// TwinCAT 3 PLC project smarAct
// Title: ESO LDC SmarAct Library
// Company: ESO
// Author: Dan Popovic
// ProjectVersion: 0.0.2.1
// Description: Local Device Control - LDC SmarAct Library based on State Machine.
// ProgramVersion: 3.1.4023.0
// libraries:
//   ESO LDC Comm Common Library, * (ESO)
//   ESO LDC Comm Tcp Library, * (ESO)
//   Tc2_Standard, * (Beckhoff Automation GmbH)
//   Tc2_System, * (Beckhoff Automation GmbH)
//   Tc2_TcpIp, * (Beckhoff Automation GmbH)
//   Tc2_Utilities, * (Beckhoff Automation GmbH)
//   Tc3_Module, * (Beckhoff Automation GmbH)
//   VisuDialogs, * (System)
//   VisuSymbols,3.5.10.0,System
// project tree:
//   DUTs/Enumerated/ E_SA_CH_ERROR.TcDUT, E_SA_RPC_ERROR.TcDUT, E_SA_POS_ELT_STATE.TcDUT, E_SA_POS_ELT_SUBSTATE.TcDUT, E_SA_CH_CMD.TcDUT, E_SA_CH_STATE.TcDUT, E_SA_CMD_TYPE.TcDUT, E_SA_DEV_STATE.TcDUT, E_SA_MOD_STATE.TcDUT, E_SA_POS_SM_STATE.TcDUT
//   DUTs/Simulation/ E_SA_SIM_CH_SM_STATE.TcDUT, T_SA_SIM_CH_CFG.TcDUT, T_SA_SIM_CH_CTRL.TcDUT, T_SA_SIM_CH_STATUS.TcDUT
//   DUTs/Structures/ T_SA_CFG.TcDUT, T_SA_CH_CFG.TcDUT, T_SA_CH_CTRL.TcDUT, T_SA_CH_STATUS.TcDUT, T_SA_CH_STATE.TcDUT, T_SA_COMMAND.TcDUT, T_SA_CTRL.TcDUT, T_SA_DEV_STATUS.TcDUT, T_SA_MOD_STATE.TcDUT, T_SA_DEV_STATE.TcDUT, T_SA_STATUS.TcDUT
//   Examples/ FB_SA_CH_PDS_IRIS.TcPOU, FB_SMARACT_SIM.TcPOU, FB_SMARACT_PDS.TcPOU
//   / GlobalTextList.TcGTLO, PlcTask.TcTTO, Visualization Manager.TcVMO (not stored)
//   POUs/ FB_SMAR_ACT_BASE.TcPOU, FB_SA_CHANNEL_BASE.TcPOU, F_GetRpcErrorText.TcPOU, F_STRING_TO_LINT.TcPOU, MAIN.TcPOU
//   POUs/Simulation/ FB_SIM_SA_CHANNEL.TcPOU, FB_SIM_SMAR_ACT.TcPOU
//   Version/ Global_Version.TcGVL
//   VISUs/GUIs/ GUI_SmarAct_PDS.TcVIS, GUI_SmarAct_SIM.TcVIS
//   VISUs/Templates/ GUI_TEMPLATE_SMAR_ACT.TcVIS
// real-time tasks:
//   TASK PlcTask: cycle T#1ms, priority 20, ADS port 350
// I/O:
//   DEVICE Device 1 (EtherCAT), AmsNetId 134.171.12.217.2.1
//     Term 1 (EK1200) [EK1200-5000 EtherCAT Power supply (2A E-Bus)]
//       Term 2 (EL6002) [EL6002 Interface 2Ch. (RS232)]
//       Term 3 (EK1110) [EK1110 EtherCAT extension]
//     Term 4 (EK1100) [EK1100 EtherCAT Coupler (2A E-Bus)]
//       Term 5 (EL3068) [EL3068 8Ch. Ana. Input 0-10V]
//       Term 6 (EL4008) [EL4008 8Ch. Ana. Output 0-10V, 12bit]
//       Term 7 (EL2008) [EL2008 8Ch. Dig. Output 24V, 0.5A]
//       Term 8 (EL1008) [EL1008 8Ch. Dig. Input 24V, 3ms]
//       Term 9 (EL3202) [EL3202 2Ch. Ana. Input PT100 (RTD)]
//       Term 10 (EL6614) [EL6614 4 Port Switch (Ethernet, CoE)]
//       Term 11 (EL6688) [EL6688 - External Synchronisation Interface (IEEE1588)]
//       Term 12 (EL9011) [EL9011 End Terminal]
// variable links:
//   smarAct/smarAct Instance <-> Device 1 (EtherCAT)/Term 4 (EK1100)/Term 10 (EL6614)
//     PlcTask Inputs/MAIN.SIM_SA.Device.i_nCouplerState <-> InfoData/State
//     PlcTask Inputs/MAIN.SmarAct_PDS.comm.i_nCouplerState <-> InfoData/State
//     PlcTask Inputs/MAIN.SmarAct_Sim.comm.i_nCouplerState <-> InfoData/State
//   smarAct/smarAct Instance <-> Device 1 (EtherCAT)/Term 4 (EK1100)/Term 8 (EL1008)
//     PlcTask Inputs/MAIN.i_bDummy <-> Channel 1/Input

CONFIGURATION smarAct
    RESOURCE PLC ON TwinCAT3
        TASK PlcTask(INTERVAL := T#1ms, PRIORITY := 20);
        PROGRAM MAIN WITH PlcTask : MAIN;
    END_RESOURCE
END_CONFIGURATION

// ---- DUTs/Enumerated/E_SA_CH_ERROR.TcDUT
{attribute 'qualified_only'}
// 'strict' cannot be used since we mix our own codes with TC codes
//{attribute 'strict'}
TYPE E_SA_CH_ERROR :
(
	OK				:= 0,
	HW_NOT_OP,
	CONFIG,				// Configuration problem, e.g. pointers not set.		
	LOCAL,			
	SETPOS,
	STOP,
	
	ABORT,
	SW_LIMIT_LOWER,
	SW_LIMIT_UPPER,
	ENABLE,
	CTRL,				// MCS2 controller error
	COMM				// MCS2 controller communication problem

);
END_TYPE

// ---- DUTs/Enumerated/E_SA_RPC_ERROR.TcDUT
{attribute 'qualified_only'}
//{attribute 'strict'}
TYPE E_SA_RPC_ERROR :
(
	OK						:= 0,
	NOT_OP					:= -1,			
	NOT_NOTOP_READY			:= -2,			
	NOT_NOTOP_NOTREADY		:= -3,			
	LOCAL					:= -4,			
	SW_LIMIT_LOWER			:= -5,			
	SW_LIMIT_UPPER			:= -6,			
	CHANNEL					:= -7,			
	VEL_ZERO				:= -8,			
	VEL_NEG					:= -9,			
	VEL_MAX					:= -10,			
	CH_NOT_OP				:= -11,
	CTRL_ERROR				:= -12,
	MOVING					:= -13,
	COMM					:= -14	// MCS2 Controller communication problem			
);
END_TYPE

// ---- DUTs/Enumerated/E_SA_POS_ELT_STATE.TcDUT
{attribute 'qualified_only'}
{attribute 'strict'}
TYPE E_SA_POS_ELT_STATE :
(
	NONE	:= 0,
	NOTOP,
	OP
);
END_TYPE

// ---- DUTs/Enumerated/E_SA_POS_ELT_SUBSTATE.TcDUT
{attribute 'qualified_only'}
{attribute 'strict'}
TYPE E_SA_POS_ELT_SUBSTATE :
(
	NONE					:= 0,
	
	NOTOP_NOTREADY			:= 100,
	NOTOP_READY				:= 101,
	NOTOP_INITIALIZING		:= 102,
	NOTOP_ABORTING			:= 107,
	
	NOTOP_ERROR				:= 199,
	
	
	OP_STANDSTILL			:= 216,            
	OP_MOVING				:= 217,
	OP_SETTING_POS			:= 218,
	OP_STOPPING				:= 219,
	
	OP_ERROR				:= 299
);
END_TYPE

// ---- DUTs/Enumerated/E_SA_CH_CMD.TcDUT
{attribute 'qualified_only'}
{attribute 'strict'}
TYPE E_SA_CH_CMD :
(
	NONE	:= 0,
	RESET,
	CALIB,
	REF,
	ENABLE,
	DISABLE,
	STOP,
	MOV
);
END_TYPE

// ---- DUTs/Enumerated/E_SA_CH_STATE.TcDUT
{attribute 'qualified_only'}
{attribute 'strict'}
TYPE E_SA_CH_STATE :
(
	BIT_ACTIVELY_MOVING			:=	16#00000001,
	BIT_CLOSED_LOOP_ACTIVE		:=	16#00000002,
	BIT_CALIBRATING				:=	16#00000004,
	BIT_REFERENCING				:=	16#00000008,
	BIT_MOVE_DELAYED			:=	16#00000010,
	BIT_SENSOR_PRESENT			:=	16#00000020,
	BIT_IS_CALIBRATED			:=	16#00000040,
	BIT_IS_REFERENCED			:=	16#00000080,
	BIT_END_STOP_REACHED		:=	16#00000100,
	BIT_RANGE_LIMIT_REACHED		:=	16#00000200,
	BIT_FOLLOWING_LIMIT_REACHED	:=	16#00000400,
	BIT_MOVEMENT_FAILED			:=	16#00000800,
	BIT_IS_STREAMING			:=	16#00001000,
	BIT_POSITIONER_OVERLOAD		:=	16#00002000,
	BIT_OVER_TEMPERATURE		:=	16#00004000,
	BIT_REFERENCE_MARK			:=	16#00008000,
	BIT_IS_PHASED				:=	16#00010000,
	BIT_POSITIONER_FAULT		:=	16#00020000,
	BIT_AMPLIFIER_ENABLED		:=	16#00040000,
	BIT_IN_POSITION				:=	16#00080000
) UDINT;
END_TYPE

// ---- DUTs/Enumerated/E_SA_CMD_TYPE.TcDUT
{attribute 'qualified_only'}
{attribute 'strict'}
TYPE E_SA_CMD_TYPE :
(
	INIT := 0,	// Commands for system initialisation
	READ,		// Commands for Reading status
	CFG,		// Commands for Configuring channels
	CTRL		// Commands for Controlling positioners, e.g. CAL, REF, MOVE, STOP
);
END_TYPE

// ---- DUTs/Enumerated/E_SA_DEV_STATE.TcDUT
{attribute 'qualified_only'}
{attribute 'strict'}
TYPE E_SA_DEV_STATE :
(
	BIT_HM_PRESENT				:= 16#00000001,
	BIT_MOVEMENT_LOCKED			:= 16#00000002,
	BIT_AMPLIFIER_LOCKED		:= 16#00000004,
	BIT_IO_MODULE_INPUT			:= 16#00000008,
	BIT_GLOBAL_INPUT			:= 16#00000010,
	BIT_INTERNAL_COMM_FAILURE	:= 16#00000100,
	BIT_IS_STREAMING			:= 16#00001000
) UDINT;
END_TYPE

// ---- DUTs/Enumerated/E_SA_MOD_STATE.TcDUT
{attribute 'qualified_only'}
{attribute 'strict'}
TYPE E_SA_MOD_STATE :
(
	BIT_SM_PRESENT				:= 16#00000001,
	BIT_BOOSTER_PRESENT			:= 16#00000002,
	BIT_ADJUSTMENT_ACTIVE		:= 16#00000004,
	BIT_IOM_PRESENT				:= 16#00000008,
	BIT_INTERNAL_COMM_FAILURE	:= 16#00000100,
	BIT_FAN_FAILURE				:= 16#00000800,
	BIT_POWER_SUPPLY_FAILURE	:= 16#00001000,
	BIT_POWER_SUPPLY_OVERLOAD	:= 16#00002000,
	BIT_OVER_TEMPERATURE		:= 16#00004000
) UDINT;
END_TYPE

// ---- DUTs/Enumerated/E_SA_POS_SM_STATE.TcDUT
{attribute 'qualified_only'}
{attribute 'strict'}
TYPE E_SA_POS_SM_STATE :
(
	// Positioner State Machine States
	NOT_READY := 0,	// The system just started.
	CALIB,			// The Positioner is Calibrating
	INIT,			// The Positioner is INITialising/REFerencing
	POST_INIT,		// In POST_INIT we calibrate REF and read CFG once.
	CALIB_REF,		// Calibrate REF position.
	READY,			// NOT OPERATIONAL / READY (i.e. REFerenced)
	
	OP,				// Positioner is Operational
	MOVING,			// Positioner is moving
	STOP,			// Positioner is stopping
	ERROR			// Positioner is in error
);
END_TYPE

// ---- DUTs/Simulation/E_SA_SIM_CH_SM_STATE.TcDUT
{attribute 'qualified_only'}
{attribute 'strict'}
TYPE E_SA_SIM_CH_SM_STATE :
(
	IDLE := 0,
	CALIB,
	REF,
	MOV,
	STOP
);
END_TYPE

// ---- DUTs/Simulation/T_SA_SIM_CH_CFG.TcDUT
TYPE T_SA_SIM_CH_CFG :
STRUCT
	
	//
	// SmarAct Positioner configuration parameters.
	// All units are Positioner System Units [DevU], pd and nm.
	//
	
	//
	// Channel Number [0..17]
	//
	nCHAN:			UINT := 0;

	//
	// MODule number that the channel belongs to [0..5].
	//
	nMOD:			UINT;	// Module  number [0..5]

	nCLIN:			DINT := 1;	// Channel Control Loop Input (1 = SENSOR)

	nBASE_UNIT:		DINT := 2;	// Channel Base Unit (2=meter, 3=degree)

	nBASE_RES:		DINT := -9;	// Channel Base Resolution

	nTUN_MTYP:		DINT := 0;	// Channel Positioner Movement Type (0=linear, 1=rotary)

	nTUN_RTYP:		DINT := 2;	// Channel Positioner Reference Type (1=end stop, 2=single coded)

	//
	// Positioning
	//

	// Position of Reference [UU].
	// This is the position to set for the REFerence (INIT).
	// Equivalent to 'Calibrate on Switch' in FB_MOTOR.
	// ':CHAN#:POS <pos>'	
	//
	lnREF_POS:		LINT := 0;
	
	lnREF_VEL:		LINT := 1;	// Velocity for referencing DevU/s]

	lnVEL:			LINT := 1;	// Velocity for referencing DevU/s]
	
	// Hold Time [ms].
	// In-position holding time. (-1) means indefinite.
	// ':CHAN#:HOLD <time>'
	//
	nHOLD:			DINT := -1;
	

	
	// In Position Threshold in [UU].
	// ':CHAN#:INP:THR <thr>'
	//
	nINP_THR:		UDINT := 1;	
	
	// In Position Delay [ms]
	// ':CHAN#:INP:DEL <delay>'
	// Move is complete after the positioner has been in position for <delay> ms.
	//
	nINP_DEL:		UDINT := 1000;
	
	// Range Limit Min (lower limit) [UU].
	// ':CHAN#:RLIM:MIN <lim>'
	// Note: If both lrRangeLimitMin and lrRangeLimitMax are set to 0.0,
	//       limits are not set.
	//
	lnRLIM_MIN:		LINT := 0;

	// Range Limit Max (upper limit) [UU].
	// ':CHAN#:RLIM:MAX <lim>'
	//
	lnRLIM_MAX:		LINT := 0;


	//
	// Calibration, Referencing (INIT) and State configuration
	//
	
	// Referencing Options.
	// :CHAN#:REF:OPT <opt>
	// It is expected that only the direction for referencing is needed to be configured.
	//    0 – positive (default)
	//    1 - negative
	nREF_OPT:		UINT := 0;

	// Calibration Options.
	// :CHAN#:CAL:OPT <opt>
	// It is expected that only the direction for Calibration is needed to be configured.
	//    0 – positive (default)
	//    1 - negative
	nCAL_OPT:		UINT := 0;

	// Positionign control options.
	// 256 - ‘In Position’ flag is set on move completion.
	// ':CHAN#:PCON:OPT <opt>'
	nPCON_OPT:		UINT := 256;
	
	
	
END_STRUCT
END_TYPE

// ---- DUTs/Simulation/T_SA_SIM_CH_CTRL.TcDUT
TYPE T_SA_SIM_CH_CTRL :
STRUCT
	
	nMode:	DINT := 0;		// Movement type: 0 - Absolute, 1 - Relative. 
	lnPOS:	LINT;			// Position in Positioner/Device Units, i.e. [nd] or [pm]
	lnVEL:	LINT := 1000;	// Velocity in Positioner/Device, i.e. [nd/s] or [pm/s]
	
END_STRUCT
END_TYPE

// ---- DUTs/Simulation/T_SA_SIM_CH_STATUS.TcDUT
TYPE T_SA_SIM_CH_STATUS :
STRUCT
	//
	// Positioner State Machine State.
	// Depending on the State, different command sets will be executed.
	//
	nPosState:			E_SA_POS_SM_STATE := E_SA_POS_SM_STATE.NOT_READY;
	

	//
	// Channel Configuration parameters read from the controller.
	// A channel is a Positioner.
	//
	nCLIN:				DINT;			// Control Loop Input, 1-SENSOR
	nTUN_BASE_UNIT:		DINT;			// Positioner Base Unit, 2-meter, 3-degree
	nTUN_BASE_RES:		DINT;			// Positioner Base Resolution, 1x10-9 or 1x10-12
	nTUN_MTYP:			DINT;			// Positioner Movement Type, 0-linear, 1-rotation, etc
	nTUN_RTYP:			DINT;			// Positioner Reference Type, 2-SINGLE_CODED


	lnPosTarget:		LINT;			// Target  position in Positioner Units
	lnPosActual:		LINT;			// Current position in Positioner Units
	lnPosStart:			LINT;			// Starting position for MOVE in Positioner Units
	lnDistance:			LINT := 0;		// move distance


	bConfigured:		BOOL;			// Flag if M_Configure has been executed.	
	bError:				BOOL;
	bInitialised:		BOOL;			// Flag if positioner has been initialised/referenced

	//
	// Channel State parameters read from the controller
	// A channel is a Positioner.
	//
	nSTATE:				UDINT;			// Positioner State as UDINT
	stState:			T_SA_CH_STATE;	// Positioner State structure, from nSTATE
	
END_STRUCT
END_TYPE

// ---- DUTs/Structures/T_SA_CFG.TcDUT
TYPE T_SA_CFG EXTENDS T_RS_BASE_CFG:
STRUCT
	//
	// INIT commands.
	// Executed during Initialisation, before going to OPERATIONAL.
	//
	{attribute 'OPC.UA.DA' := '0'}
	cmdList_Init:	ARRAY [0..7] OF T_SA_COMMAND := [
							(cmd := '*IDN?', 			nReplies := 1),
							(cmd := ':DEV:SNUM?', 		nReplies := 1),
							(cmd := ':DEV:STAT?', 		nReplies := 1),
							(cmd := '', 		nReplies := 0),
							(cmd := '', 		nReplies := 0),
							(cmd := '', 		nReplies := 0),
							(cmd := '', 		nReplies := 0),
							(cmd := '', 		nReplies := 0)];

	//
	// List of commands to SET Channel/Positioner Configuration.
	// Note the # and *** characters !!!
	// The actual command will be set like this:
	//    #   will be replaced with channel number
	//    *** will be replaced with a value
	// Example:
	//    ':CHAN#:PCON:OPT ***' => ':CHAN1:PCON:OPT 256'
	//
	// Important NOTE:
	// At this stage RLIM:MIN and RLIM:MAX are disabled, i.e. = 0.
	// The actual limits will be set at the E_SA_POS_SM_STATE.CALIB_REF stage,
	// see M_SetCmdList().
	//
	// These commands are sent only once, just before the positioner is 
	// commanded to Reference (INIT).
	//
	{attribute 'OPC.UA.DA' := '0'}
	cmdList_CfgSet:	ARRAY [0..15] OF T_SA_COMMAND := [
							(cmd := ':CHAN#:CAL:OPT ***', 		nReplies := 0),
							(cmd := ':CHAN#:REF:OPT ***', 		nReplies := 0),
							(cmd := ':CHAN#:PCON:OPT ***', 		nReplies := 0),
							(cmd := ':CHAN#:HOLD ***', 			nReplies := 0),
							(cmd := ':CHAN#:INP:THR ***', 		nReplies := 0),
							(cmd := ':CHAN#:INP:DEL ***', 		nReplies := 0),
							(cmd := ':CHAN#:RLIM:MIN 0', 		nReplies := 0),
							(cmd := ':CHAN#:RLIM:MAX 0', 		nReplies := 0),
							(cmd := ':CHAN#:VEL ***', 			nReplies := 0),
							(cmd := ':REF#', 					nReplies := 0),
							(cmd := '', 		nReplies := 0),
							(cmd := '', 		nReplies := 0)];
							

	//				
	// List of commands to GET Channel/Positioner Configuration.
	// These commands are sent from the moment the SW started till the positioner 
	// has been Calibrated or Referenced (INIT).
	// Once the Positioer is Ready, these commans are not sent any more.
	//
	{attribute 'OPC.UA.DA' := '0'}
	cmdList_POST_INIT:	ARRAY [0..15] OF T_SA_COMMAND := [
							(cmd := ':MOD#:STAT?', 			nReplies := 1),
							(cmd := ':CHAN#:STAT?', 		nReplies := 1),
							(cmd := ':CHAN#:CAL:OPT?', 		nReplies := 1),
							(cmd := ':CHAN#:REF:OPT?', 		nReplies := 1),
							(cmd := ':CHAN#:PCON:OPT?', 	nReplies := 1),
							(cmd := ':CHAN#:INP:THR?', 		nReplies := 1),
							(cmd := ':CHAN#:INP:DEL?', 		nReplies := 1),
							(cmd := ':CHAN#:RLIM:MIN?', 	nReplies := 1),
							(cmd := ':CHAN#:RLIM:MAX?', 	nReplies := 1),
							(cmd := ':CHAN#:POS:TARG?', 	nReplies := 1),
							(cmd := ':CHAN#:POS:CURR?', 	nReplies := 1),
							(cmd := '', 		nReplies := 0),
							(cmd := '', 		nReplies := 0),
							(cmd := '', 		nReplies := 0),
							(cmd := '', 		nReplies := 0),
							(cmd := '', 		nReplies := 0)];
							

	//
	// List of Monitoring commands in PRE-OPERATION.
	// Executed before the Positioner has been Referenced/initialised.
	//
	{attribute 'OPC.UA.DA' := '0'}
	cmdList_NOT_READY:	ARRAY [0..15] OF T_SA_COMMAND := [
							(cmd := ':MOD#:STAT?', 			nReplies := 1),
							(cmd := ':CHAN#:STAT?', 		nReplies := 1),
							(cmd := ':CHAN#:POS:TARG?', 	nReplies := 1),
							(cmd := ':CHAN#:POS:CURR?', 	nReplies := 1),
							(cmd := ':CHAN#:PCON:OPT?', 	nReplies := 1),
							(cmd := ':CHAN#:CLIN?', 		nReplies := 1),
							(cmd := ':CHAN#:TUN:BASE:UNIT?',nReplies := 1),
							(cmd := ':CHAN#:TUN:BASE:RES?', nReplies := 1),
							(cmd := ':CHAN#:TUN:MTYP?', 	nReplies := 1),
							(cmd := ':CHAN#:TUN:RTYP?', 	nReplies := 1),
							(cmd := ':CHAN#:INP:THR?', 		nReplies := 1),
							(cmd := ':CHAN#:INP:DEL?', 		nReplies := 1),
							(cmd := ':CHAN#:RLIM:MIN?', 	nReplies := 1),
							(cmd := ':CHAN#:RLIM:MAX?', 	nReplies := 1),
							(cmd := '', 		nReplies := 0),
							(cmd := '', 		nReplies := 0)];
			

	//
	// List of Monitoring commands in OPERATION.
	// Executed once the Positioner has been Referenced/initialised.
	//
	{attribute 'OPC.UA.DA' := '0'}
	cmdList_Mon:	ARRAY [0..15] OF T_SA_COMMAND := [
							(cmd := ':MOD#:STAT?', 			nReplies := 1),
							(cmd := ':CHAN#:STAT?', 		nReplies := 1),
							(cmd := ':CHAN#:POS:TARG?', 	nReplies := 1),
							(cmd := ':CHAN#:POS:CURR?', 	nReplies := 1),
							(cmd := '', 		nReplies := 0),
							(cmd := '', 		nReplies := 0),
							(cmd := '', 		nReplies := 0),
							(cmd := '', 		nReplies := 0),
							(cmd := '', 		nReplies := 0),
							(cmd := '', 		nReplies := 0),
							(cmd := '', 		nReplies := 0),
							(cmd := '', 		nReplies := 0),
							(cmd := '', 		nReplies := 0),
							(cmd := '', 		nReplies := 0),
							(cmd := '', 		nReplies := 0),
							(cmd := '', 		nReplies := 0)];
			

	//
	// Array of used channels. Set to TRUE for each used channel.
	// 18 channels max. 6 modules [0..5], 3 connections each [CH1, CH2, CH3].
	// channel = (Module x 3) + (CH-1)
	// For example:
	//   First connection (CH1) of first module (Module0): channel = 0 x 3 + (1-1) = 0
	//   Second connection (CH2) of first module (Module0): channel = 0 x 3 + (2-1) = 1
	//   Third connection (CH3) of third module (Module2): channel = 2 x 3 + (3-1) = 8
	//  
	arrUsedCh:	ARRAY [0..17] 	OF BOOL;	

	//
	// Array of used modules. Set to TRUE for each used module.
	// Automatically populated in method M_Configure().
	//
	arrUsedMod:	ARRAY [0..5] 	OF BOOL;	
	
	// Channel configuration structures
//	arrChCfg:	ARRAY [0..17] OF T_SA_CH_CFG;

END_STRUCT
END_TYPE

// ---- DUTs/Structures/T_SA_CH_CFG.TcDUT
TYPE T_SA_CH_CFG :
STRUCT
	sName:	STRING := 'Not Used';	// Positioner name, e.g. 'PYR Filter Wheel'
	sUnits:	STRING := 'none';		// Positioner User Units
	
	bUsed:	BOOL;
	
	lrMaxVelocity:	LREAL := 1.0;	// Maximum velocity	[UU]
	
	//
	// SmarAct Positioner configuration parameters.
	// All units are User Units [UU], mm, deg, etc.
	// The driver converts them into Positioner units.
	// During Referencing (INIT), these parameters will be written to
	// the positioner.
	// The monitoring task will read them from the positioner and 
	// save them into T_SA_CH_STATUS that is contained in T_SA_STATUS.
	//
	
	//
	// Channel Number [0..17]
	//
	// 18 channels max. 6 modules [0..5], 3 connections each [CH1, CH2, CH3].
	// channel = (Module x 3) + (CH-1)
	// For example:
	//   First connection (CH1) of first module (Module0): channel = 0 x 3 + (1-1) = 0
	//   Second connection (CH2) of first module (Module0): channel = 0 x 3 + (2-1) = 1
	//   Third connection (CH3) of third module (Module2): channel = 2 x 3 + (3-1) = 8
	//  
	nCHAN:			UINT := 0;

	//
	// MODule number that the channel belongs to [0..5].
	// Calculated from the channel number. i.e. the index of this instance.
	// channel = (Module x 3) + (CH-1)
	// Module = index / 3
	// index = 0, 1 or 2    => Module = 0
	// index = 3, 4 or 5    => Module = 1
	// ...
	// index = 15, 16 or 17 => Module = 5
	//
	nMOD:			UINT;	// Module  number [0..5]

	//
	// Positioning
	//

	// Conversion from UU to SmarAct units, i.e. [nd] or [pm].
	// This is just the correction of the Base Resolution (if needed).
	// Pos [SmarAct] = lnScale * Pos [UU] / EXPT(10, T_SA_CH_STATUS:nTUN_BASE_RES)
	//
	lrScale:		LREAL := 1.0;	
	
	
	// Position of Reference [UU].
	// This is the position to set for the REFerence (INIT).
	// Equivalent to 'Calibrate on Switch' in FB_MOTOR.
	// Set position for Reference in User Units
	// ':CHAN#:POS <pos>'	
	// <pos> = lrREF_POS  / EXPT(10, T_SA_CH_STATUS:nTUN_BASE_RES) * lnScale
	//
	lrREF_POS:		LREAL := 0;
	
	lrREF_VEL:		LREAL := 0.01;	// Velocity for referencing [UU/s]
	
	// Hold Time [ms].
	// In-position holding time. (-1) means indefinite.
	// ':CHAN#:HOLD <time>'
	//
	nHOLD:			DINT := -1;
	
	
	
	// In Position Threshold in [UU].
	// ':CHAN#:INP:THR <thr>'
	//
	lrINP_THR:		LREAL := 0.01;	
	
	// In Position Delay [ms]
	// ':CHAN#:INP:DEL <delay>'
	// Move is complete after the positioner has been in position for <delay> ms.
	//
	nINP_DEL:		UDINT := 1000;
	
	// Range Limit Min (lower limit) [UU].
	// ':CHAN#:RLIM:MIN <lim>'
	// Note: If both lrRangeLimitMin and lrRangeLimitMax are set to 0.0,
	//       limits are not set.
	//
	lrRangeLimitMin:	LREAL := 0.0;

	// Range Limit Max (upper limit) [UU].
	// ':CHAN#:RLIM:MAX <lim>'
	//
	lrRangeLimitMax:	LREAL := 0.0;
	
	
	//
	// Calibration, Referencing (INIT) and State configuration
	//
	
	// Referencing Options.
	// :CHAN#:REF:OPT <opt>
	// It is expected that only the direction for referencing is needed to be configured.
	//    0 – positive (default)
	//    1 - negative
	nREF_OPT:		UINT := 0;

	// Calibration Options.
	// :CHAN#:CAL:OPT <opt>
	// It is expected that only the direction for Calibration is needed to be configured.
	//    0 – positive (default)
	//    1 - negative
	nCAL_OPT:		UINT := 0;

	// Positionign control options.
	// 256 - ‘In Position’ flag is set on move completion.
	// ':CHAN#:PCON:OPT <opt>'
	nPCON_OPT:		UINT := 256;
	
	
	
END_STRUCT
END_TYPE

// ---- DUTs/Structures/T_SA_CH_CTRL.TcDUT
TYPE T_SA_CH_CTRL :
STRUCT
	//
	// Control structure for a single channel/positioner.
	//
	
	//
	// Active command.
	// Setting nCmd to something other than NONE will
	// trigger execution of commands REF, STOP, MOV.
	//
	nCmd:	E_SA_CH_CMD := E_SA_CH_CMD.NONE;	// Active command

	lrPos:	LREAL;		// Position in User Units, i.e. [deg] or [mm]
	lrOff:	LREAL;		// Position offset in User Units, i.e. [deg] or [mm]
	lrVel:	LREAL;		// Velocity in User Units, i.e. [deg/s] or [mm/sec]
	
END_STRUCT
END_TYPE

// ---- DUTs/Structures/T_SA_CH_STATUS.TcDUT
TYPE T_SA_CH_STATUS :
STRUCT
	bLocal:			BOOL	:= FALSE;	// if TRUE, device operated from PLC GUI 

	nErrorCode: 	E_SA_CH_ERROR 	:= E_SA_CH_ERROR.OK;	// Error code 
	nRpcErrorCode: 	E_SA_RPC_ERROR 	:= E_SA_RPC_ERROR.OK;	// RPC Error code

	bCtrlCommProblem:	BOOL;			// SmarAct MCS2 Controller Comm Problem
	nCtrlErrorCode: E_SM_ERROR;			// SmarAct MCS2 Controller Error code
	nCtrlState:		E_RS_BASE_STATE;	// SmarAct MCS2 Controller State	

	sErrorText: 	STRING 	:= 'OK'; 			// Error text 
	sRpcErrorText: 	STRING 	:= 'OK'; 			// RPC Error text 
	sStatus: 		STRING 	:= 'OK'; 			// Status in textual form, e.g. 'OFF' 
	
	//
	// Standard ELT States and Substates
	//
	nState:			E_SA_POS_ELT_STATE 		:= E_SA_POS_ELT_STATE.NOTOP;
	nSubstate:		E_SA_POS_ELT_SUBSTATE	:= E_SA_POS_ELT_SUBSTATE.NOTOP_NOTREADY;
	
	sState:			STRING	:= 'NOTOP';
	sSubstate:		STRING	:= 'NOT READY';

	//
	// Positioner State Machine State.
	// Depending on the State, different command sets will be executed.
	//
	nPosState:			E_SA_POS_SM_STATE := E_SA_POS_SM_STATE.NOT_READY;
	nLastPosState:		E_SA_POS_SM_STATE := E_SA_POS_SM_STATE.NOT_READY;
	

	lrPosTarget:		LREAL;			// Target  position in User Units
	lrPosActual:		LREAL;			// Current position in User Units

	bConfigured:		BOOL;			// Flag if M_Configure has been executed.	
	bError:				BOOL;
	bEnabled:			BOOL;			// Flag if axis is enabled
	bInitialised:		BOOL;			// Flag if positioner has been initialised/referenced
	bInPosition:		BOOL;			// Flag if axis is In-Position

	//
	// Channel State parameters read from the controller
	// A channel is a Positioner.
	//
	nCH_STATE:				UDINT;			// Positioner State as UDINT
	{attribute 'OPC.UA.DA' := '0'}
	stState:			T_SA_CH_STATE;	// Positioner State structure, from nSTATE
	
	//
	// Device/Channel/Positioner status in user units, i.e. [pm] and [nd].
	// These values are read periodically.
	// Values are normally huge, e.g. pos=18000000000 [nd].
	//
	{attribute 'OPC.UA.DA' := '0'}
	devStatus:			T_SA_DEV_STATUS; 	
	
END_STRUCT
END_TYPE

// ---- DUTs/Structures/T_SA_CH_STATE.TcDUT
TYPE T_SA_CH_STATE :
STRUCT
	//
	// Channel State
	// Got with the ':CHAN#:STAT?' command
	//
	bACTIVELY_MOVING:			BOOL;
	bCLOSED_LOOP_ACTIVE:		BOOL;
	bCALIBRATING:				BOOL;
	bREFERENCING:				BOOL;
	bMOVE_DELAYED:				BOOL;
	bSENSOR_PRESENT:			BOOL;
	bIS_CALIBRATED:				BOOL;
	bIS_REFERENCED:				BOOL;
	bEND_STOP_REACHED:			BOOL;
	bRANGE_LIMIT_REACHED:		BOOL;
	bFOLLOWING_LIMIT_REACHED:	BOOL;
	bMOVEMENT_FAILED:			BOOL;
	bIS_STREAMING:				BOOL;
	bPOSITIONER_OVERLOAD:		BOOL;
	bOVER_TEMPERATURE:			BOOL;
	bREFERENCE_MARK:			BOOL;
	bIS_PHASED:					BOOL;
	bPOSITIONER_FAULT:			BOOL;
	bAMPLIFIER_ENABLED:			BOOL;
	bIN_POSITION:				BOOL;

	bERROR:						BOOL := TRUE;
	
END_STRUCT
END_TYPE

// ---- DUTs/Structures/T_SA_COMMAND.TcDUT
TYPE T_SA_COMMAND :
STRUCT
	cmd:		STRING := '';	(* Command to send *)
	nReplies:	UINT;   		(* Number of replies, i.e. reply terminators *)
END_STRUCT
END_TYPE

// ---- DUTs/Structures/T_SA_CTRL.TcDUT
TYPE T_SA_CTRL EXTENDS T_RS_BASE_CTRL :
STRUCT
	// Arrays of structures for Configuration and Control commands.
	// Note that only one positioner is handled in each monitoring cycle.
	{attribute 'OPC.UA.DA' := '0'}
	cmdList:			ARRAY [0..15]	OF T_SA_COMMAND;	// List of up to 16 Commands per channel
	
END_STRUCT
END_TYPE

// ---- DUTs/Structures/T_SA_DEV_STATUS.TcDUT
//
// Device/Channel/Positioner status in user units, i.e. [pm] and [nd]
//
TYPE T_SA_DEV_STATUS :
STRUCT
	nCAL_OPT:			DINT;			// Calibration option
	nREF_OPT:			DINT;			// Referencing option
	nPCON_OPT:			DINT;			// Positioner Control Options, 256-'in-pos' flag
	nCLIN:				DINT;			// Control Loop Input, 1-SENSOR
	nTUN_BASE_UNIT:		DINT;			// Positioner Base Unit, 2-meter, 3-degree
	nTUN_BASE_RES:		DINT;			// Positioner Base Resolution, 1x10-9 or 1x10-12
	nTUN_MTYP:			DINT;			// Positioner Movement Type, 0-linear, 1-rotation, etc
	nTUN_RTYP:			DINT;			// Positioner Reference Type, 2-SINGLE_CODED
	nINP_THR:			DINT;			// In Position Threshold [DevU]
	nINP_DEL:			DINT;			// In Position Delay [ms]
	nRLIM_MIN:			LINT;			// MIN Limit [DevU]
	nRLIM_MAX:			LINT;			// MAX Limit [DevU]

	lnPosTarget:		LINT;			// Target  position in Positioner Units
	lnPosActual:		LINT;			// Current position in Positioner Units

END_STRUCT
END_TYPE

// ---- DUTs/Structures/T_SA_MOD_STATE.TcDUT
TYPE T_SA_MOD_STATE :
STRUCT
	bSM_PRESENT:			BOOL;
	bBOOSTER_PRESENT:		BOOL;
	bADJUSTMENT_ACTIVE:		BOOL;
	bIOM_PRESENT:			BOOL;
	bINTERNAL_COMM_FAILURE:	BOOL;
	bFAN_FAILURE:			BOOL;
	bPOWER_SUPPLY_FAILURE:	BOOL;
	bPOWER_SUPPLY_OVERLOAD:	BOOL;
	bOVER_TEMPERATURE:		BOOL;
	
	bInitialised:			BOOL;	// If TRUE, the state has been read from the controller.
	bUsed:					BOOL;
	bERROR:					BOOL;
END_STRUCT
END_TYPE

// ---- DUTs/Structures/T_SA_DEV_STATE.TcDUT
TYPE T_SA_DEV_STATE :
STRUCT
	bHM_PRESENT:			BOOL;
	bMOVEMENT_LOCKED:		BOOL;
	bAMPLIFIER_LOCKED:		BOOL;
	bIO_MODULE_INPUT:		BOOL;
	bGLOBAL_INPUT:			BOOL;
	bINTERNAL_COMM_FAILURE:	BOOL;
	bIS_STREAMING:			BOOL;

	bInitialised:			BOOL;	// If TRUE, the state has been read from the controller.
	bERROR:					BOOL;
END_STRUCT
END_TYPE

// ---- DUTs/Structures/T_SA_STATUS.TcDUT
TYPE T_SA_STATUS EXTENDS T_RS_BASE_STAT :
STRUCT
	nNumMod:		UINT;			// Total number of MODules [0..6]. Should be >= 1.
	nNumCh:			UINT;			// Total number of CHannels [0..18]. Should be >= 1.

	nRetries:		UDINT := 0;		// Total number of retries in case of communication problems
	
	sLibVersion:	STRING	:= 'UNKNOWN';		// Library version as string, e.g. '1.2.0.0'
	sReply:			STRING(255); 	// Last device Reply to predefined commands
	lastCtrlCmd:	STRING;			// Last Ctrl command sent to Device
	
	nDevState:		UDINT;
	sIDN:			STRING := '';	// Device info
	sDevSerNum:		STRING := '';	// Device serial number
	
	{attribute 'OPC.UA.DA' := '0'}
	stDevState:		T_SA_DEV_STATE;						// DEVice state
	
	{attribute 'OPC.UA.DA' := '0'}
	arrModState:	ARRAY [0..5]  OF T_SA_MOD_STATE;	// Array of MODule state
	
END_STRUCT
END_TYPE

// ---- Version/Global_Version.TcGVL
{attribute 'TcGenerated'}
{attribute 'no-analysis'}
{attribute 'linkalways'}
// This function has been automatically generated from the project information.
VAR_GLOBAL CONSTANT
	{attribute 'const_non_replaced'}
	stLibVersion_ESO_LDC_SmarAct_Library : ST_LibVersion := (iMajor := 0, iMinor := 0, iBuild := 2, iRevision := 1, nFlags := 0, sVersion := '0.0.2.1');
END_VAR

// ---- POUs/MAIN.TcPOU
PROGRAM MAIN
VAR
	//
	// TcpIp related variables.
	// Mandatory for all PLC programs using TcpIp !!!
	// On PLC reset or program download close all existing connections.
	//
    fbSocketCloseAll:	FB_SocketCloseAll;
    bCloseAll: 			BOOL := TRUE;
	bAllCosed:			BOOL := FALSE;

	//
	// Devices
	//
	{attribute 'OPC.UA.DA' := '1'}
	SmarAct_PDS:		FB_SMARACT_PDS;		// SmarAct Device for PDS
	{attribute 'OPC.UA.DA' := '1'}
	SmarAct_Sim:		FB_SMARACT_SIM;		// Simulated SmarAct

	//
	// Simulators
	//
	SIM_SA:				FB_SIM_SMAR_ACT;	// SmarAct simulator
	
	i_bDummy	AT %I*:	BOOL;	// Dummy var to get System OPERATIONAL without I/O
	
END_VAR

//
// Mandatory for all PLC programs using TcpIp !!!
// On PLC reset or program download close all existing connections.
//
IF NOT bAllCosed	THEN
	IF bCloseAll THEN
		bCloseAll := FALSE;
		fbSocketCloseAll( sSrvNetId:= '', bExecute:= TRUE, tTimeout:= T#10s );
	ELSE
		fbSocketCloseAll( bExecute:= FALSE );
	END_IF
	
	IF fbSocketCloseAll.bBusy THEN
		RETURN;
	ELSE
		bAllCosed	:= TRUE;
	END_IF
END_IF



//
// SmarAct Controller Instance PDS
//
SmarAct_PDS(
	in_sName			:= 'SmarAct PDS',
	in_bSimulation		:= FALSE,
	in_nPeriod			:= 300,				// Delay between channels 300ms = 0.3s
	in_sCmdSuffix		:= '$0D$0A',		// Command terminator '[CR][LF]'='$0D$0A'
	in_sReplySuffix		:= '$0D$0A',		// Reply terminator '[CR][LF]'='$0D$0A'
	in_sDeviceTcpIpAdr	:= '192.168.1.200',	// Device IP address
	in_nDeviceTcpPort	:= 55551);


//
// SmarAct Controller Instance SIMulated
//
SmarAct_Sim(
	in_sName			:= 'SmarAct SIM',
	in_bSimulation		:= TRUE,
	in_nPeriod			:= 500,				// Delay between channels 500ms = 0.5s
	in_sCmdSuffix		:= '$0D$0A',		// Command terminator '[CR][LF]'='$0D$0A'
	in_sReplySuffix		:= '$0D$0A',		// Reply terminator '[CR][LF]'='$0D$0A'
	in_sDeviceTcpIpAdr	:= '127.0.0.1',		// Simulated device IP address. MUST be '127.0.0.1' !!!
	in_nDeviceTcpPort	:= 55551);


//
// SmarAct simulator that communicates with SmarAct_Sim.
// It should not exist in real PLC application.
// Not that in simulation the IP MUST be '127.0.0.1' !!!
//
SIM_SA(
	in_bSimulation:= TRUE, 
	in_bEnable:= TRUE, 
	in_sReplySuffix:= '$0D$0A', 
	in_sTcpIpAdr:= '127.0.0.1',	// Simulator IP address, 
	in_nTcpPort:= 55551);

END_PROGRAM

// ---- Examples/FB_SMARACT_PDS.TcPOU
FUNCTION_BLOCK FB_SMARACT_PDS EXTENDS FB_SMAR_ACT_BASE
VAR_INPUT
END_VAR
VAR_OUTPUT
END_VAR
VAR
	//
	// TODO USER: Add existing SmarAct Positioners.
	//
	// We use prefix 'x_' just for the convenience that
	// all positioners appear together in the OPC UA Namespace.
	//
	x_fw:		FB_SA_CHANNEL_BASE;	// CH 0
	x_iris:		FB_SA_CH_PDS_IRIS;	// CH 1 non-linear scaling for % of opening
END_VAR

//
// Execute the base class object FB_SMAR_ACT_BASE.
//
SUPER^();

METHOD M_ConfigureUser
VAR_INPUT
END_VAR
//
// This method defines specific configurations for 
// each positioner/channel in PDS.
//


// 
// In this example, two positioners are defined in FB_SMARACT_PDS.
//
//	fw:		FB_SA_CHANNEL_BASE;	// CH 0
//	iris:	FB_SA_CHANNEL_BASE;	// CH 1
//

//
// Configure used channels [0..17].
// There are two used channels: 0 and 1.
//
cfg.arrUsedCh[0]	:= TRUE;
cfg.arrUsedCh[1]	:= TRUE;


//
// Set pointers to instances of used channels
//
ptrCH[0]	:= ADR(x_fw);
ptrCH[1]	:= ADR(x_iris);


//
// Initial configuration of each exiting positioner.
//

//
// SFW-6-25.4 - Filter Wheel
//
x_fw.M_Configure(
	in_sName			:= 'PYR Filter Wheel',
	in_sUnits			:= 'deg',
	in_lrScale			:= 1.0, 
	in_lrREF_POS		:= 0.0,		// REF mark pos
	in_lrREF_VEL		:= 20.0,	// Velocity for referencing [UU/s]
	in_nHOLD			:= -1,		// Hold infinitely
	in_lrINP_THR		:= 0.001,	// in-pos threshold = 0.001 deg
	in_nINP_DEL			:= 500,		// in-pos delay 500 ms
	in_lrMaxVelocity	:= 30,		// Maximum permitted Velocity
	in_lrRangeLimitMin	:= 0.0,		// Min=Max ==> No limits
	in_lrRangeLimitMax	:= 0.0,		// Min=Max ==> No limits 
	in_nREF_OPT			:= 0,		// Referencing in positive direction
	in_nCAL_OPT			:= 0,		// Calibrating in positive direction
	in_nPCON_OPT		:= 256);	// 'in-pos' flag set

//
// SID-50 - Iris Diaphragm
//
// Note: Because the scale is negative, MIN and MAX values are swapped.
//       In Device Units, the diaphragm will move between -5..-50 (/scale) mm.
//       In User   Units, the diaphragm will move between 1..100 %.
//
// The position of the diaphragm is the percentage of the opening.
//

x_iris.M_Configure(
	in_sName			:= 'SHAPS Diaphragm',
	in_sUnits			:= '%',
	in_lrScale			:= -0.001763245, 
	in_lrREF_POS		:= 34.33,	// REF mark pos in %. (Diam = 29.29832067 mm)
	in_lrREF_VEL		:= 5.0,		// Velocity for referencing [UU/s]
	in_nHOLD			:= -1,		// Hold infinitely
	in_lrINP_THR		:= 0.0005,	// in-pos threshold = 0.0005 %
	in_nINP_DEL			:= 500,		// in-pos delay 500 ms
	in_lrMaxVelocity	:= 15,		// Maximum permitted Velocity
	in_lrRangeLimitMin	:= 100.001,	// Min limit (positive because in_lrScale < 0) !!!
	in_lrRangeLimitMax	:= 0.999,	// Max limit (negative because in_lrScale < 0) !!!
	in_nREF_OPT			:= 0,		// Referencing in positive direction
	in_nCAL_OPT			:= 0,		// Calibrating in positive direction
	in_nPCON_OPT		:= 256);	// 'in-pos' flag set
END_METHOD

END_FUNCTION_BLOCK

// ---- POUs/FB_SMAR_ACT_BASE.TcPOU
FUNCTION_BLOCK FB_SMAR_ACT_BASE EXTENDS FB_RS_BASE
VAR_INPUT
	{attribute 'OPC.UA.DA' := '0'}
	in_bAutoMonitor:	BOOL := TRUE;	// If true, it starts PERIODIC reads (monitoring) after INIT
	{attribute 'OPC.UA.DA' := '0'}
	in_nPeriod:			DINT := 1000;	// Interval for periodic reading [ms], default 1000 ms = 1 sec
	{attribute 'OPC.UA.DA' := '0'}
	in_sCmdSuffix:		STRING(16);		// Terminator for command: LS336 '$0A', LS224 '$0D$0A'
	{attribute 'OPC.UA.DA' := '0'}
	in_sReplySuffix:	STRING(16);		// Terminator for reply

	{attribute 'OPC.UA.DA' := '0'}
	in_sDeviceTcpIpAdr: STRING(16);		// Device IP address, e.g. '192.168.0.80'
	{attribute 'OPC.UA.DA' := '0'}
    in_nDeviceTcpPort:	UINT;			// Device Tcp port, default 7777 
END_VAR
VAR_OUTPUT
END_VAR
VAR
	{attribute 'OPC.UA.DA' := '1'}
	cfg:		T_SA_CFG;	
	{attribute 'OPC.UA.DA' := '1'}
	ctrl:		T_SA_CTRL;	

	{attribute 'OPC.UA.DA' := '1'}
	{attribute 'OPC.UA.DA.Access' := '1'}
	stat:		T_SA_STATUS;	(* Common State Machine Status - ReadOnly *)

	//
	// Pointers for up to 18 channels/positioners.
	// They are defined in FBs that EXTEND FB_SMAR_ACT_BASE.
	//
	{attribute 'OPC.UA.DA' := '0'}
	ptrCH:	ARRAY [0..17] OF POINTER TO FB_SA_CHANNEL_BASE;
	
	//
	// Array of up to 18 channel/positioner names.
	// Needed for GUI automation in case of uninitialised pointers.
	//
	{attribute 'OPC.UA.DA' := '0'}
	arrChName:	ARRAY [0..17] OF STRING;
	
	{attribute 'OPC.UA.DA' := '0'}
	nGuiIndex:	UINT;	// Index of Positioner to display on GUI
	
	// Pointer to Channel instance to be diplayed on GUI.
	// Set in M_SetGuiPointer().
	ptrGuiCH:	POINTER TO FB_SA_CHANNEL_BASE;	
	
	// Communication interface is added for any FB derived from FB_RS_BASE.
	// That's why we need pointers, e.g. ptrReadCmds.
	// We also need pointers to structures inside FB_RS_COMM, e.g. ptrCommCfg.
	{attribute 'OPC.UA.DA' := '0'}
	ptrCommCfg:		POINTER TO T_RS_COMM_CFG;	(* Pointer to comm.cfg instance *)
	{attribute 'OPC.UA.DA' := '0'}
	ptrCommCtrl:	POINTER TO T_RS_COMM_CTRL;	(* Pointer to comm.ctrl instance *)
	{attribute 'OPC.UA.DA' := '0'}
	ptrCommStat:	POINTER TO T_RS_COMM_STAT;	(* Pointer to comm.stat instance *)


	(* Timers *)
	{attribute 'OPC.UA.DA' := '0'}
	fbTimer:		TON; (* General Timeout *)

	(* Misc internal vars *)
	{attribute 'OPC.UA.DA' := '0'}
	cmdCounter:		INT := 1;	// Position in commands table
	{attribute 'OPC.UA.DA' := '0'}
	bResult:		BOOL := FALSE;


	{attribute 'OPC.UA.DA' := '0'}
	comm:		FB_TCP_CLIENT;			// Instance of Tcp comm FB. OPC UA Disabled!!!
	
	
	
END_VAR

//
//	Configure the device.
// This will set proper references and pointers.
//
M_Configure();


//
// Execute comm instance.
//
comm(	in_bSimulation		:= in_bSimulation,
		in_sDeviceTcpIpAdr	:= in_sDeviceTcpIpAdr,
		in_nDeviceTcpPort	:= in_nDeviceTcpPort, 
		in_sCmdSuffix		:= in_sCmdSuffix, 
		in_sReplySuffix		:= in_sReplySuffix,
		in_nPollingDelay 	:= 50,
		in_nTimeout			:= 2000);


//
// Execute the base class object FB_RS_BASE.
//
SUPER^();


//
// Pass the SmarAct MCS2 Controller error status to
// all positioners under its control.
//
M_PassCtrlState();


//
// Set pointer to Channel instance to be displayed on GUI.
//
M_SetGuiPointer();

METHOD ActivityInitializing
VAR_INPUT
	bExecute:	BOOL;
END_VAR
VAR_INST
	{attribute 'OPC.UA.DA' := '0'}
    nMethodState:	INT := 0;	// State Machine current state
END_VAR
SetAction('ActivityInitializing');


IF NOT bExecute THEN
	nMethodState	:= 0;	// Reset the state machine
	cmdCounter		:= -1;	// First init command. CASE 15: will increment it to 0
	RETURN;
END_IF

// Handle State Machine
CASE nMethodState OF
	0:	// Initialize COMM port
		(* Reset the port *)
		ptrCommCtrl^.nCommand	:= E_RS_COMM_CMD.INIT;
		ptrCommCtrl^.bExecute	:= TRUE;

		(* Start the timer by going false/true *)
		fbTimer (IN := FALSE); (* Reset timer *)
		fbTimer (IN := TRUE, PT := T#5S); (* 5 sec timeout for reply *)

		nMethodState 	:= 15;	// On next cycle wait until the comm port is reset, i.e. idle
		
	15:	// Wait IDLE
		fbTimer (IN := TRUE);
		IF M_GetCommStatus() = E_RS_COMM_STATUS.IDLE  AND M_GetCommInitialised() THEN
			// Communication is IDLE 
			fbTimer (IN := FALSE);	// disable timer 
			stat.sReply		:= ptrCommStat^.sReply;	// Save the reply

			// Extract values from the reply to a stat variable.
			IF ptrCommCtrl^.bHasReply	THEN
				// Index is not important for INIT commands because they don't
				// refer to MODule or CHANnel.
				// We put zero for the input parameter.
				M_ReadFromReply(0);	// Index is not important for INIT commands.
			END_IF

			cmdCounter		:= cmdCounter + 1;	// Increment init command index
			fbTimer (IN := FALSE);	// disable timer 
			fbTimer (IN := TRUE, PT := cfg.tDelay_Init); // Wait INIT delay
			bCommProblem	:= FALSE;
			nMethodState 	:= 18;	// Execute next device INIT command
		ELSIF M_GetCommStatus() = E_RS_COMM_STATUS.ERROR  AND fbTimer.ET > T#4900MS THEN
			fbTimer (IN := FALSE);
			SetStatus(E_LAKESHORE_ERROR.COMM, 'ERROR: Communication error');	
			bCommProblem	:= TRUE;
			nEvent := E_SM_EVENT.ERRINIT;
			RETURN;
		ELSIF fbTimer.Q THEN
			// Timer expired after 5 sec. This is an error.
			fbTimer (IN := FALSE);
			SetStatus(E_LAKESHORE_ERROR.TIMEOUT, 'ERROR: Communication timeout');	
			bCommProblem	:= TRUE;
			nEvent := E_SM_EVENT.ERRINIT;
			RETURN;
		END_IF

	
	
	18:	// Wait INIT Delay
		fbTimer (IN := TRUE);
		IF fbTimer.Q THEN
			// Timer expired after 5 sec. This is an error.
			fbTimer (IN := FALSE);
			nMethodState 	:= 20;	// Execute next device INIT command
			RETURN;
		END_IF

	
	
	20:	// INIT DEV
		IF cfg.cmdList_Init[cmdCounter].cmd = '' THEN
			// Device INIT is done. Go to IDLE 
			stat.bInitialised 	:= TRUE;
			cmdCounter			:= 1;
			SetStatus(E_SM_ERROR.OK, 'IDLE');
			nEvent 		:= E_SM_EVENT.INITDONE;
			RETURN;
		END_IF
		
		(* Send INIT command with index cmdCounter *)
		ptrCommCtrl^.nCommand		:= E_RS_COMM_CMD.SEND;
		ptrCommCtrl^.sCmd			:= cfg.cmdList_Init[cmdCounter].cmd;
		ptrCommCtrl^.nNumReplies	:= cfg.cmdList_Init[cmdCounter].nReplies;
		ptrCommCtrl^.bHasReply		:= cfg.cmdList_Init[cmdCounter].nReplies > 0;
		ptrCommCtrl^.bExecute		:= TRUE;
	
		(* Start the timer by going false/true *)
		fbTimer (IN := FALSE); (* Reset timer *)
		fbTimer (IN := TRUE, PT := T#5S); (* 5 sec timeout for reply *)

		// On next cycle wait until the comm port is idle
		nMethodState 	:= 15;	// On next cycle wait until the comm port is idle
	
END_CASE
END_METHOD

METHOD ActivityMonitoring
VAR_INPUT
	bExecute:	BOOL;
END_VAR
VAR_INST
	{attribute 'OPC.UA.DA' := '0'}
    nMethodState:	INT := 0;	// State Machine current state
	{attribute 'OPC.UA.DA' := '0'}
	nRetries:		INT := 0;	// Number of retries in case of communication problems
	{attribute 'OPC.UA.DA' := '0'}
	nCmdType:		E_SA_CMD_TYPE := E_SA_CMD_TYPE.READ;
	{attribute 'OPC.UA.DA' := '0'}
	devCmd:			T_SA_COMMAND;	// Device command to be sent
	
	// TODO: Testing
	{attribute 'OPC.UA.DA' := '0'}
	nChIdx:			UINT := 0;	// Channel index for testing of hash character handling
	{attribute 'OPC.UA.DA' := '0'}
	nCmdIdx:		UINT := 0;	// Command index in specific command list. [0..15]

END_VAR
//
// At least one module must be used.
// If not, don't do anything.
//
IF stat.nNumMod = 0	THEN
	SetAction('ERROR: No Module Used !!!'); 
	SetStatus(E_SM_ERROR.INIT_FAILURE, 'ERROR: No Module Used !!!');
	RETURN;
END_IF

IF NOT cfg.bAutoMonitor AND stat.nSubstate = E_RS_BASE_SUBSTATE.NOTOP_READY THEN
	SetAction('No Monitoring'); 
	SetStatus(E_SM_ERROR.OK, 'IDLE');
	nMethodState	:= 0;	// Reset the state machine
	RETURN;
END_IF

IF NOT bExecute THEN
	SetAction('ActivityMonitoring'); 
	SetStatus(E_SM_ERROR.OK, 'BUSY');
	nMethodState	:= 0;	// Reset the state machine
	nCmdType		:= E_SA_CMD_TYPE.READ;	// We start with READ commands.
	RETURN;
END_IF

// Handle State Machine
CASE nMethodState OF
	0:	// Get valid channel.
		// This call will check if the current channel is used.
		// If not, it will take next available channel.
		nChIdx	:= M_GetValidChannel(nChIdx);
		
		// If this is the very first command for the channel,
		// Set commands.
		IF nCmdIdx = 0	THEN
			M_SetCmdList(nChIdx);
		END_IF
		
		
		// Get next command to execute.
		// The command depends on the state of the positioner and 
		// the current index (nCmdIdx) of the command in the list.
		//
		devCmd	:= M_GetCommand(nCmdIdx);
	
			
		// Check if we have arrived at the end of the command list.
		// In this case, go to the next channel.
		IF devCmd.cmd = '' THEN
			// We have executed all commands.
			// Check if we have to exit Monitoring
			IF nNextState <> E_RS_BASE_STATE.NONE	THEN
				SetStatus(E_SM_ERROR.OK, nNextDescription);
				SetState(nNextState, nNextSubstate);
				nNextState		:= E_RS_BASE_STATE.NONE;
				nNextSubstate	:= E_RS_BASE_SUBSTATE.NONE;
				nNextDescription:= '';
				RETURN;
			END_IF

			//
			// Update Positioner status
			//
			ptrCH[nChIdx]^.M_UpdateStatus();
			
			
			// Check if the State Machine State should be changed.
			// If yes, M_SetNextPosState() will set new state and return TRUE.
			// This can happen due to any Positioner control command (CAL, REF, RESET, ENABLE, DISABLE, MOVE or STOP)
			IF ptrCH[nChIdx]^.M_SetNextPosState()	THEN
				// The State has changed.
				// Reset command index to 0, i.e. start from the first command.
				nCmdIdx	:= 0;
			ELSE
				// Get NEXT valid channel
				nChIdx	:= M_GetValidChannel(nChIdx + 1);
				
				// Reset command index to 0
				nCmdIdx	:= 0;
			END_IF
						
				
			// Wait tDelay_Periodic before re-starting the READ.
			SetStatus(E_SM_ERROR.OK, 'IDLE');
			
			(* Start the timer by going false/true *)
			fbTimer (IN := FALSE); (* Reset timer *)
			fbTimer (IN := TRUE, PT := cfg.tDelay_Periodic);
			nMethodState 	:= 10;	// Goto Wait for tDelay_Periodic
			RETURN;
		END_IF
		
		// Send command
		ptrCommCtrl^.nCommand		:= E_RS_COMM_CMD.SEND;
		ptrCommCtrl^.sCmd			:= devCmd.cmd;
		ptrCommCtrl^.nNumReplies	:= devCmd.nReplies;
		ptrCommCtrl^.bHasReply		:= devCmd.nReplies > 0;
		ptrCommCtrl^.bExecute		:= TRUE;
		
		
		
		statRef.sErrorText	:= 'BUSY';

		// In case we are executing a CTRL command with no replies,
		// we apply a long timeout.
		// However, when the comm port becomes IDLE and after at 
		// least 200ms, we go to the next command. (see nMethodState 12:)
		IF NOT ptrCommCtrl^.bHasReply THEN
			fbTimer (IN := FALSE); // Reset timer
			fbTimer (IN := TRUE, PT := T#10S); 
			nCmdIdx			:= nCmdIdx + 1;	// Go to next command.
			nMethodState	:= 12;				// Goto WAIT for delay
			RETURN;
		ELSE			
			// There is a reply, i.e. this is a 'READ' command.
			// For regular READ commands, apply short delay of 10ms before 
			// checking the status of comm port. 
			// Start the timer by going false/true
			fbTimer (IN := FALSE); // Reset timer
			fbTimer (IN := TRUE, PT := T#10MS);	

			statRef.sErrorText	:= 'BUSY';
			nMethodState := 15;	// Goto short delay
			RETURN;
		END_IF
		
		
		
	10:	// Wait until the delay timeout expires
		fbTimer (IN := TRUE);

		(* If Timer has expired, go to the next state. *)
		IF fbTimer.Q THEN
			fbTimer (IN := FALSE);
			nMethodState 	:= 0;				// Goto handling of next command
			RETURN;
		END_IF
	
	12:	// Wait until the comm port is idle and at least 200ms have expired.
		// Otherwise, wait the PT period.
		fbTimer (IN := TRUE);

		IF (M_GetCommStatus() = E_RS_COMM_STATUS.IDLE  AND  fbTimer.ET > T#200MS)	OR
			fbTimer.Q	THEN
			fbTimer (IN := FALSE);
			nMethodState 	:= 0;				// Goto handling of next command
			RETURN;
		END_IF

	
	15:	// Wait until the delay timeout expires
		fbTimer (IN := TRUE);

		(* If Timer has expired, go to the next state. *)
		IF fbTimer.Q THEN
			fbTimer (IN := FALSE);
			fbTimer (IN := TRUE, PT := T#3S);	// 3 sec timeout for reply
			statRef.sErrorText	:= 'BUSY';
			nMethodState 	:= 20;	// Goto Wait for IDLE/Reply
			RETURN;
		END_IF
	



	20:	// Wait for the reading to complete, i.e. IDLE
		fbTimer (IN := TRUE);
		IF M_GetCommStatus() = E_RS_COMM_STATUS.IDLE THEN
			// Communication is IDLE 
			fbTimer (IN := FALSE);	// disable timer 
			stat.sReply		:= ptrCommStat^.sReply;	// Save the reply
			
			// Extract values from the reply to a stat variable.
			M_ReadFromReply(nChIdx);

			bCommProblem	:= FALSE;
			nRetries		:= 0;	// Reset number of retries

			nCmdIdx			:= nCmdIdx + 1;	// Go to next command.
			
			nMethodState 	:= 0;				// Goto Send command
			nEvent := E_SM_EVENT.COMMOK;
			RETURN;
		ELSIF M_GetCommStatus() = E_RS_COMM_STATUS.ERROR OR fbTimer.Q THEN
			fbTimer (IN := FALSE);
			SetStatus(E_LAKESHORE_ERROR.COMM, 'ERROR: Communication error');	
			bCommProblem	:= TRUE;
			// Retry up to 2 times
			nRetries		:= nRetries + 1;		// Increment number of retries
			stat.nRetries	:= stat.nRetries + 1;	// Increment total number of retries
			IF nRetries > 1 THEN
				nEvent := E_SM_EVENT.ERRCOMM;
				RETURN;
			END_IF
			// Apply a short delay of 1 sec and retry
			fbTimer (IN := FALSE); (* Reset timer *)
			fbTimer (IN := TRUE, PT := T#1000MS);
			nMethodState := 10;				// Goto Wait 
			RETURN;
		END_IF

	
END_CASE
END_METHOD

METHOD M_Configure
VAR_INPUT
END_VAR
VAR
	i:		UINT;
	nMod:	UINT;	// Module number
END_VAR
//
// NOTE: Do not touch this method.
//       Specific configuration is given in M_ConfigureUser().
//

IF NOT stat.bConfigured	THEN
	
	// Set references - MANDATORY !!!
	cfgRef	REF=cfg;
	ctrlRef	REF=ctrl;
	statRef	REF=stat;
	
	
	// Copy timeouts from the input parameters
	cfg.tDelay_Periodic	:= DINT_TO_TIME(in_nPeriod);
	cfg.tDelay_Ctrl		:= T#50MS;

	
	// Assign list of commands to read before Positioner is initialised
	ctrl.cmdList		:= cfg.cmdList_NOT_READY;
	
	
	// Set pointers to comm, i.e.
	ptrCommCfg	:= ADR(comm.cfg);	(* Pointer to comm.cfg instance *)
	ptrCommCtrl	:= ADR(comm.ctrl);	(* Pointer to comm.ctrl instance *)
	ptrCommStat	:= ADR(comm.stat);	(* Pointer to comm.stat instance *)
	

	// Set comm suffixes for commands and replies
	ptrCommCfg^.sCmdSuffix		:= in_sCmdSuffix;
	ptrCommCfg^.sReplySuffix	:= in_sReplySuffix;

	
	//
	// Execute specific user configuration.
	// This method configures all used channels.
	//
	M_ConfigureUser();
	

	//
	// Set bUsed flag, channel and module number for each used Channel. 
	// Populate array of Used Modules.
	//
	FOR i:=0 TO 17 DO
		IF cfg.arrUsedCh[i]	= TRUE	THEN
			IF ptrCH[i] = 0	THEN
				// Check if pointers are correctly set.
				stat.sErrorText := 'ERROR: Pointer to FB_SA_CHANNEL_BASE not set!'; 
				RETURN;
			END_IF
			ptrCH[i]^.M_SetChannel(i);
			// Get module number
			nMod	:= ptrCH[i]^.M_GetModule();
			// Set MOD bUsed flag 
			stat.arrModState[nMod].bUsed 	:= TRUE;
			cfg.arrUsedMod[nMod] 			:= TRUE;
			// Set GUI label
			arrChName[i]	:= ptrCH[i]^.cfg.sName;
		ELSE
			arrChName[i]	:= 'Not Used';
		END_IF
	END_FOR
	
	
	//
	// Get the total number of Modules
	//
	stat.nNumMod	:= 0;
	FOR i:=0 TO 5 DO
		IF stat.arrModState [i].bUsed	THEN
			stat.nNumMod	:= stat.nNumMod + 1;
		END_IF
	END_FOR
	

	//
	// Get the total number of Channels
	//
	stat.nNumCh	:= 0;
	FOR i:=0 TO 17 DO
		IF cfg.arrUsedCh[i]	THEN
			stat.nNumCh	:= stat.nNumCh + 1;
		END_IF
	END_FOR
	
	
	// Get the smarAct.library version 
	stat.sLibVersion	:= stLibVersion_ESO_LDC_SmarAct_Library.sVersion;


	// Configuration completed
	stat.bConfigured	:= TRUE;
END_IF
END_METHOD

METHOD M_ConfigureUser
VAR_INPUT
END_VAR
//
// This is an example of method M_ConfigureUser() that
// must be provided for each customized FB that EXTENDS the 
// functionality of FB_SMAR_ACT_BASE.
// The method defines specific configurations for each positioner/channel.
//

//
// TODO USER
//

// 
// In the following example, it is assumed that there are two positioners defined
// In the FB that EXTENDS FB_SMAR_ACT_BASE. (see FBs in Examples directory)
//
// 	fw:		FB_SA_CHANNEL_BASE;
//	iris:	FB_SA_CHANNEL_BASE;
//


//
// Set used channels [0..17].
// In this example, we use channels 0 and 1.
//
(*
cfg.arrUsedCh[0]	:= TRUE;
cfg.arrUsedCh[1]	:= TRUE;
*)


//
// Set pointers to instances of used channels
//
(*
ptrCH[0]	:= ADR(fw);
ptrCH[1]	:= ADR(iris);
*)



/////////////////////////////////////////////////////////////
// Specific configuration for each SmarAct Channel/Positioner
/////////////////////////////////////////////////////////////
(*
//
// SFW-6-25.4 - Filter Wheel, Channel 0
//
fw.M_Configure(
	in_sName			:= 'PYR Filter Wheel',
	in_lrScale			:= 1.0, 
	in_lrREF_POS		:= 0.0,		// REF mark pos
	in_lrREF_VEL		:= 20.0,	// Velocity for referencing [UU/s]
	in_nHOLD			:= -1,		// Hold infinitely
	in_lrINP_THR		:= 0.001,	// in-pos threshold = 0.001 deg
	in_nINP_DEL			:= 500,		// in-pos delay 500 ms
	in_lrMaxVelocity	:= 30,		// Maximum permitted Velocity
	in_lrRangeLimitMin	:= 0.0,		// Min=Max ==> No limits
	in_lrRangeLimitMax	:= 0.0,		// Min=Max ==> No limits 
	in_nREF_OPT			:= 0,		// Referencing in positive direction
	in_nCAL_OPT			:= 0,		// Calibrating in positive direction
	in_nPCON_OPT		:= 256);	// 'in-pos' flag set

//
// SID-50 - Iris Diaphragm, Channel 1
//
iris.M_Configure(
	in_sName			:= 'SHAPS Diaphragm',
	in_lrScale			:= -0.000772, 
	in_lrREF_POS		:= 25.244,	// REF mark pos
	in_lrREF_VEL		:= 5.0,		// Velocity for referencing [UU/s]
	in_nHOLD			:= -1,		// Hold infinitely
	in_lrINP_THR		:= 0.0002,	// in-pos threshold = 0.0002 UU
	in_nINP_DEL			:= 500,		// in-pos delay 500 ms
	in_lrMaxVelocity	:= 20,		// Maximum permitted Velocity
	in_lrRangeLimitMin	:= 0.0,		// Min limit
	in_lrRangeLimitMax	:= 0.0,		// Max limit 
	in_nREF_OPT			:= 0,		// Referencing in positive direction
	in_nCAL_OPT			:= 0,		// Calibrating in positive direction
	in_nPCON_OPT		:= 256);	// 'in-pos' flag set
*)
END_METHOD

METHOD M_GetChMod : UINT
VAR_INPUT
	index:	UINT;
END_VAR
M_GetChMod	:= ptrCH[index]^.M_GetModule();
END_METHOD

//
// Get command with index 'index' from ctrl.cmdList[]
//
METHOD M_GetCommand : T_SA_COMMAND
VAR_INPUT
	index:		UINT;
END_VAR
VAR
	emptyCmd:	T_SA_COMMAND;
END_VAR
IF index < 0 OR index > 15	THEN
	// The index is not valid. Set empty command.
	M_GetCommand	:= emptyCmd;
ELSE
	M_GetCommand	:= ctrl.cmdList[index];
END_IF
END_METHOD

METHOD M_GetCommInitialised : BOOL
VAR_INPUT
END_VAR
// This is just a dummy method for BASE FB
M_GetCommInitialised	:= comm.M_GetInitialised();
END_METHOD

METHOD M_GetCommStatus : E_RS_COMM_STATUS
VAR_INPUT
END_VAR
M_GetCommStatus	:= comm.M_GetStatus();
END_METHOD

METHOD M_GetDevState
VAR_INPUT
	nStatus:	UDINT;
END_VAR
stat.stDevState.bHM_PRESENT				:= UDINT_TO_BOOL(nStatus AND E_SA_DEV_STATE.BIT_HM_PRESENT);
stat.stDevState.bMOVEMENT_LOCKED			:= UDINT_TO_BOOL(nStatus AND E_SA_DEV_STATE.BIT_MOVEMENT_LOCKED);
stat.stDevState.bAMPLIFIER_LOCKED		:= UDINT_TO_BOOL(nStatus AND E_SA_DEV_STATE.BIT_AMPLIFIER_LOCKED);
stat.stDevState.bIO_MODULE_INPUT			:= UDINT_TO_BOOL(nStatus AND E_SA_DEV_STATE.BIT_IO_MODULE_INPUT);
stat.stDevState.bGLOBAL_INPUT			:= UDINT_TO_BOOL(nStatus AND E_SA_DEV_STATE.BIT_GLOBAL_INPUT);
stat.stDevState.bINTERNAL_COMM_FAILURE	:= UDINT_TO_BOOL(nStatus AND E_SA_DEV_STATE.BIT_INTERNAL_COMM_FAILURE);
stat.stDevState.bIS_STREAMING			:= UDINT_TO_BOOL(nStatus AND E_SA_DEV_STATE.BIT_IS_STREAMING);

IF	stat.stDevState.bHM_PRESENT				OR
	stat.stDevState.bMOVEMENT_LOCKED			OR
	stat.stDevState.bAMPLIFIER_LOCKED		OR
	stat.stDevState.bINTERNAL_COMM_FAILURE	OR
	stat.stDevState.bIS_STREAMING				THEN
	stat.stDevState.bERROR	:= TRUE;
ELSE
	stat.stDevState.bERROR	:= FALSE;
END_IF
END_METHOD

METHOD M_GetModStatus
VAR_INPUT
	index:		UINT;
	nStatus:	UDINT;
END_VAR
// MODule index is [0..5]
IF index > 5	THEN
	RETURN;
END_IF

stat.arrModState[index].bSM_PRESENT				:= UDINT_TO_BOOL(nStatus AND E_SA_MOD_STATE.BIT_SM_PRESENT);
stat.arrModState[index].bBOOSTER_PRESENT		:= UDINT_TO_BOOL(nStatus AND E_SA_MOD_STATE.BIT_BOOSTER_PRESENT);
stat.arrModState[index].bADJUSTMENT_ACTIVE		:= UDINT_TO_BOOL(nStatus AND E_SA_MOD_STATE.BIT_ADJUSTMENT_ACTIVE);
stat.arrModState[index].bIOM_PRESENT			:= UDINT_TO_BOOL(nStatus AND E_SA_MOD_STATE.BIT_IOM_PRESENT);
stat.arrModState[index].bINTERNAL_COMM_FAILURE	:= UDINT_TO_BOOL(nStatus AND E_SA_MOD_STATE.BIT_INTERNAL_COMM_FAILURE);
stat.arrModState[index].bFAN_FAILURE			:= UDINT_TO_BOOL(nStatus AND E_SA_MOD_STATE.BIT_FAN_FAILURE);
stat.arrModState[index].bPOWER_SUPPLY_FAILURE	:= UDINT_TO_BOOL(nStatus AND E_SA_MOD_STATE.BIT_POWER_SUPPLY_FAILURE);
stat.arrModState[index].bPOWER_SUPPLY_OVERLOAD	:= UDINT_TO_BOOL(nStatus AND E_SA_MOD_STATE.BIT_POWER_SUPPLY_OVERLOAD);
stat.arrModState[index].bOVER_TEMPERATURE		:= UDINT_TO_BOOL(nStatus AND E_SA_MOD_STATE.BIT_OVER_TEMPERATURE);

IF	stat.arrModState[index].bINTERNAL_COMM_FAILURE	OR
	stat.arrModState[index].bFAN_FAILURE			OR
	stat.arrModState[index].bPOWER_SUPPLY_FAILURE	OR
	stat.arrModState[index].bPOWER_SUPPLY_OVERLOAD	OR
	stat.arrModState[index].bOVER_TEMPERATURE			THEN
		stat.arrModState[index].bERROR	:= TRUE;
ELSE
		stat.arrModState[index].bERROR	:= FALSE;
END_IF
END_METHOD

METHOD M_GetRpcErrorText : STRING
VAR_INPUT
	ErrorCode:	INT;
END_VAR
VAR
	str:	STRING;
END_VAR
CASE ErrorCode OF
	E_SA_RPC_ERROR.OK:					str	:= 'OK';
	E_SA_RPC_ERROR.NOT_OP:				str	:= 'Not initialised, i.e. not in channel OP state.';
	E_SA_RPC_ERROR.NOT_NOTOP_READY:		str	:= 'Call failed. Not in NOTOP_READY.';
	E_SA_RPC_ERROR.NOT_NOTOP_NOTREADY:	str	:= 'Call failed. Not in NOTOP_NOTREADY/ERROR.';
	E_SA_RPC_ERROR.LOCAL:				str	:= 'RPC calls not allowed in Local mode.';
	E_SA_RPC_ERROR.SW_LIMIT_LOWER:		str	:= 'Target position beyond Lower SW Limit';
	E_SA_RPC_ERROR.SW_LIMIT_UPPER:		str	:= 'Target position beyond Upper SW Limit';
	E_SA_RPC_ERROR.CHANNEL:				str	:= 'Channel not in range [0..17]';
	E_SA_RPC_ERROR.VEL_MAX:				str	:= 'Target Velocity higher than Maximum';
	E_SA_RPC_ERROR.VEL_NEG:				str	:= 'Target Velocity cannot be negative';
	E_SA_RPC_ERROR.VEL_ZERO:			str	:= 'Target Velocity cannot be zero';
	E_SA_RPC_ERROR.CH_NOT_OP:			str	:= 'Channel not OPERATIONAL. REFerence first.';
ELSE
	str	:= 'Unregistered RPC error.';
END_CASE

M_GetRpcErrorText	:= str;
END_METHOD

METHOD M_GetValidChannel : UINT
VAR_INPUT
	index:	UINT;
END_VAR
VAR
	i:	UINT;
END_VAR
// Return first available Channel index, starting from 'index'.
// Channels are in range [0..17]
FOR i:= index TO 17 DO
	IF cfg.arrUsedCh[i] = TRUE	THEN
		M_GetValidChannel	:= i;
		RETURN;
	END_IF
END_FOR

// We didn't find any, start from zero index again.
FOR i:= 0 TO 17 DO
	IF cfg.arrUsedCh[i] = TRUE	THEN
		M_GetValidChannel	:= i;
		RETURN;
	END_IF
END_FOR
END_METHOD

METHOD M_PassCtrlState
VAR_INPUT
END_VAR
VAR
	i:	UINT;
END_VAR
FOR i:= 0 TO 17 DO
	IF ptrCH[i] <> 0	THEN
		ptrCH[i]^.M_GetCtrlState(bCommProblem, stat.nErrorCode, stat.nState);
	END_IF
END_FOR
END_METHOD

METHOD M_ReadFromReply : BOOL
VAR_INPUT
	index:	UINT;	// Channel number!
END_VAR
VAR
	pos:			INT;	// Position of the terminator in the reply.
    parsed_reply: 	STRING;
	refChStatus:	REFERENCE TO T_SA_CH_STATUS;
END_VAR
//
// Reply should always end with in_sReplySuffix ('$R$N') character.
// Otherwise, it's an error.
// Only commands with the reply from which the value should be read are handled.
//


pos := FIND (stat.sReply, in_sReplySuffix);
IF pos > 0	THEN
    parsed_reply := LEFT(stat.sReply, LEN(stat.sReply) - LEN(in_sReplySuffix));
	
	//
	// INIT commands, not related to MODule or CHANnel.
	//
	IF ptrCommCtrl^.sCmd = '*IDN?' THEN
		// Get the DEVice ID
		stat.sIDN	:= parsed_reply;
		
	ELSIF ptrCommCtrl^.sCmd = ':DEV:STAT?' THEN
		// Get the DEVice state
		stat.nDevState	:= STRING_TO_UDINT(parsed_reply);
		M_GetDevState(stat.nDevState);
		
	ELSIF ptrCommCtrl^.sCmd = ':DEV:SNUM?' THEN
		// Get the DEVice Serial Number
		stat.sDevSerNum	:= parsed_reply;

	//
	// Replies to commands starting with ':MOD'.
	//
	ELSIF FIND(ptrCommCtrl^.sCmd, ':MOD') = 1 THEN
		IF FIND(ptrCommCtrl^.sCmd, ':STAT?') > 1 THEN
			// FB_SA_CHANNEL::M_GetModule() returns the index of the MODule
			M_GetModStatus(ptrCH[index]^.M_GetModule(), STRING_TO_UDINT(parsed_reply));
		END_IF

	//
	// Replies to commands starting with ':CHAN'.
	//
	ELSIF FIND(ptrCommCtrl^.sCmd, ':CHAN') = 1  THEN
		// We need a REFerence in order to write attributes inside FB.
		refChStatus REF=ptrCH[index]^.stat;

		IF FIND(ptrCommCtrl^.sCmd, ':STAT?') > 1 THEN
			ptrCH[index]^.M_SetChanState(STRING_TO_UDINT(parsed_reply));
	
		ELSIF FIND(ptrCommCtrl^.sCmd, ':PCON:OPT?') > 1 THEN
			refChStatus.devStatus.nPCON_OPT	:= STRING_TO_DINT(parsed_reply);
	
		ELSIF FIND(ptrCommCtrl^.sCmd, ':CLIN?') > 1 THEN
			refChStatus.devStatus.nCLIN	:= STRING_TO_DINT(parsed_reply);
	
		ELSIF FIND(ptrCommCtrl^.sCmd, ':TUN:BASE:UNIT?') > 1 THEN
			refChStatus.devStatus.nTUN_BASE_UNIT	:= STRING_TO_DINT(parsed_reply);
	
		ELSIF FIND(ptrCommCtrl^.sCmd, ':TUN:BASE:RES?') > 1 THEN
			refChStatus.devStatus.nTUN_BASE_RES	:= STRING_TO_DINT(parsed_reply);
	
		ELSIF FIND(ptrCommCtrl^.sCmd, ':TUN:MTYP?') > 1 THEN
			refChStatus.devStatus.nTUN_MTYP	:= STRING_TO_DINT(parsed_reply);
	
		ELSIF FIND(ptrCommCtrl^.sCmd, ':TUN:RTYP?') > 1 THEN
			refChStatus.devStatus.nTUN_RTYP	:= STRING_TO_DINT(parsed_reply);
	
		ELSIF FIND(ptrCommCtrl^.sCmd, ':INP:THR?') > 1 THEN
			refChStatus.devStatus.nINP_THR	:= STRING_TO_DINT(parsed_reply);
	
		ELSIF FIND(ptrCommCtrl^.sCmd, ':INP:DEL?') > 1 THEN
			refChStatus.devStatus.nINP_DEL	:= STRING_TO_DINT(parsed_reply);
	
		ELSIF FIND(ptrCommCtrl^.sCmd, ':POS:TARG?') > 1 THEN
			refChStatus.devStatus.lnPosTarget	:= F_STRING_TO_LINT(parsed_reply);
	
		ELSIF FIND(ptrCommCtrl^.sCmd, ':POS:CURR?') > 1 THEN
			refChStatus.devStatus.lnPosActual	:= F_STRING_TO_LINT(parsed_reply);
	
		ELSIF FIND(ptrCommCtrl^.sCmd, ':RLIM:MIN?') > 1 THEN
			refChStatus.devStatus.nRLIM_MIN	:= F_STRING_TO_LINT(parsed_reply);

		ELSIF FIND(ptrCommCtrl^.sCmd, ':RLIM:MAX?') > 1 THEN
			refChStatus.devStatus.nRLIM_MAX	:= F_STRING_TO_LINT(parsed_reply);
		END_IF	
	END_IF	
	
	M_ReadFromReply	:= TRUE; (* OK *)
ELSE
	M_ReadFromReply	:= FALSE;	//	Failed to read from the reply
END_IF
END_METHOD

METHOD M_SetCmdList
VAR_INPUT
	index:			UINT := 0;	// Channel index
END_VAR
VAR
	nChState:	E_SA_POS_SM_STATE := ptrCH[index]^.stat.nPosState;
	i:			INT;
	cmd:		STRING;
END_VAR
//
// Copy corresponding list of commands to the list in the 'ctrl' structure.
// The generic list contains # characters !
// Examples: ':MOD#:STAT?', ':CHAN#:POS:TARG?', etc.
// They have to be replaced with Channel or Module number.
//
CASE nChState OF
	E_SA_POS_SM_STATE.NOT_READY:
		ctrl.cmdList	:= cfg.cmdList_NOT_READY;
	E_SA_POS_SM_STATE.CALIB:
		// Calibration requires only one command, ':CAL#'.
		ctrl.cmdList[0].cmd			:= ':CAL#';
		ctrl.cmdList[0].nReplies	:= 0;
		ctrl.cmdList[1].cmd			:= '';		// Command terminator
	E_SA_POS_SM_STATE.INIT:
		ctrl.cmdList	:= cfg.cmdList_CfgSet;
	E_SA_POS_SM_STATE.POST_INIT:
		ctrl.cmdList	:= cfg.cmdList_POST_INIT;
	E_SA_POS_SM_STATE.CALIB_REF:
		// First set the MIN and MAX limits.
		// Calibrate the REFerence mark. 
		// Read new MIN and MAX limits.
		ctrl.cmdList[0].cmd			:= ':CHAN#:RLIM:MIN ***';
		ctrl.cmdList[0].nReplies	:= 0;
		ctrl.cmdList[1].cmd			:= ':CHAN#:RLIM:MAX ***';
		ctrl.cmdList[1].nReplies	:= 0;
		ctrl.cmdList[2].cmd			:= ':CHAN#:POS ***';
		ctrl.cmdList[2].nReplies	:= 0;
		ctrl.cmdList[3].cmd			:= ':CHAN#:RLIM:MIN?';
		ctrl.cmdList[3].nReplies	:= 1;
		ctrl.cmdList[4].cmd			:= ':CHAN#:RLIM:MAX?';
		ctrl.cmdList[4].nReplies	:= 1;
		ctrl.cmdList[5].cmd			:= '';		// Command terminator
	E_SA_POS_SM_STATE.READY:
		ctrl.cmdList	:= cfg.cmdList_Mon;
	E_SA_POS_SM_STATE.OP:
		ctrl.cmdList	:= cfg.cmdList_Mon;
	E_SA_POS_SM_STATE.MOVING:
		// Move the positioner. 
		// Set direction ':CHAN#:VEL <vel>'
		// Set velocity ':CHAN#:VEL <vel>'
		// Move         ':MOVE# <pos>'.
		ctrl.cmdList[0].cmd			:= ':CHAN#:VEL ***';
		ctrl.cmdList[0].nReplies	:= 0;
		ctrl.cmdList[1].cmd			:= ':MOVE# ***';
		ctrl.cmdList[1].nReplies	:= 0;
		ctrl.cmdList[2].cmd			:= '';		// Command terminator
	E_SA_POS_SM_STATE.STOP:
		// Stop the positioner. 
		// Requires only one command, ':STOP#'.
		ctrl.cmdList[0].cmd			:= ':STOP#';
		ctrl.cmdList[0].nReplies	:= 0;
		ctrl.cmdList[1].cmd			:= '';		// Command terminator
	E_SA_POS_SM_STATE.ERROR:
		ctrl.cmdList	:= cfg.cmdList_Mon;
END_CASE

// Set MOD or CHAN index, depending on the command.
FOR i:=0 TO 15 DO
	cmd	:= ctrl.cmdList[i].cmd;
	IF cmd <> ''	THEN
		IF FIND(cmd, ':MOD#') = 1	THEN
			// A MODule command. Set MOD index.
			ctrl.cmdList[i].cmd			:= ptrCH[index]^.M_SetCommandModule(cmd);
		ELSIF FIND(cmd, ':CHAN#') = 1  OR  FIND(cmd, ':MOVE#') = 1	THEN
			// Channel commands.
			// Commands with parameters have the dummy string '***'.
			// Replace *** in generic command with the value.
			IF FIND(cmd, '***') > 0 THEN
				cmd	:= ptrCH[index]^.M_SetCommandValue(cmd);
			END_IF
			// Set CHAN number in the command.
			ctrl.cmdList[i].cmd			:= ptrCH[index]^.M_SetCommandChannel(cmd);
		ELSIF FIND(cmd, ':CAL#') = 1  OR  FIND(cmd, ':REF#') = 1  OR  FIND(cmd, ':STOP#') = 1	THEN
			// Channel command. Replace only the channel number.
			ctrl.cmdList[i].cmd			:= ptrCH[index]^.M_SetCommandChannel(cmd);
		END_IF
	END_IF
END_FOR
END_METHOD

METHOD M_SetGuiPointer
VAR_INPUT
END_VAR
// There are up to 18 channels [0..17].
IF nGuiIndex > 17	THEN
	nGuiIndex	:= 17;
END_IF

ptrGuiCH	:= ptrCH[nGuiIndex];
END_METHOD

METHOD ProcessEvents
VAR_INPUT
END_VAR

(* 
	Before processing the event, execute the Do-Activity tasks. 
	Note that, in case of orthogonal regions, more than one Do-Activity 
	could run in the same PLC cycle.
	Note: Most of these activities have timeouts since they take time.
*)

IF	statRef.nSubstate = E_RS_BASE_SUBSTATE.OP_MONITORING 		OR 
	statRef.nSubstate = E_RS_BASE_SUBSTATE.NOTOP_READY			OR
	(statRef.nSubstate = E_RS_BASE_SUBSTATE.NOTOP_ERROR 	AND 
	 nLastGoodSubstate = E_RS_BASE_SUBSTATE.NOTOP_READY) 		OR 
	(statRef.nSubstate = E_RS_BASE_SUBSTATE.OP_ERROR 		AND 
	 nLastGoodSubstate = E_RS_BASE_SUBSTATE.OP_MONITORING)			THEN
	ActivityMonitoring(TRUE);
ELSIF statRef.nSubstate = E_RS_BASE_SUBSTATE.NOTOP_INITIALIZING THEN
	ActivityInitializing(TRUE);
END_IF

// Set last known good substate. Used for recovery from comm problems.
M_SetLastGoodSubstate();

(* 
	Evaluate state machine transitions.
*)

CASE statRef.nState OF

//***********************************
// NOTOP
//***********************************
E_RS_BASE_STATE.NOTOP:

	(* Transitions from NOTOP substates *)
	CASE statRef.nSubstate OF
	
	E_RS_BASE_SUBSTATE.NOTOP_NOTREADY:		
		IF 	nEvent = E_SM_EVENT.INIT OR cfgRef.bAutoMonitor  THEN
			nEvent := E_SM_EVENT.INIT;
			ActionInitExecute();
			SetState(E_RS_BASE_STATE.NOTOP, E_RS_BASE_SUBSTATE.NOTOP_INITIALIZING);
			SetStatus(E_SM_ERROR.OK, 'OK');
			RETURN;
		END_IF
		
	E_RS_BASE_SUBSTATE.NOTOP_INITIALIZING:			
		IF nEvent = E_SM_EVENT.INITDONE THEN
			nReadType := E_RS_BASE_READ_TYPE.PERIODIC;
			ActivityMonitoring(FALSE);	// Reset Monitoring method
			IF cfgRef.bAutoMonitor THEN
				nEvent := E_SM_EVENT.ENABLE;
				statRef.bAutoStarted	:= TRUE;
				SetState(E_RS_BASE_STATE.OP, E_RS_BASE_SUBSTATE.OP_MONITORING);
			ELSE
				SetState(E_RS_BASE_STATE.NOTOP, E_RS_BASE_SUBSTATE.NOTOP_READY);
			END_IF
			RETURN;
		ELSIF nEvent = E_SM_EVENT.ERRINIT THEN
			// INIT failed. Keep re-trying.
			SetState(E_RS_BASE_STATE.NOTOP, E_RS_BASE_SUBSTATE.NOTOP_NOTREADY);
			RETURN;
		END_IF
		
	E_RS_BASE_SUBSTATE.NOTOP_READY:			
		IF nEvent = E_SM_EVENT.ENABLE THEN
			IF cfgRef.bAutoMonitor THEN
				// Monitoring is already in progress.
				// It has to complete the read cycle in a clean way.
				nNextState		:= E_RS_BASE_STATE.OP;					// Next state after STOP	
				nNextSubstate	:= E_RS_BASE_SUBSTATE.OP_MONITORING;	// Next substate after STOP	
				nNextDescription:= 'BUSY';
				nReadType		:= E_RS_BASE_READ_TYPE.PERIODIC;
				RETURN;
			ELSE
				SetState(E_RS_BASE_STATE.OP, E_RS_BASE_SUBSTATE.OP_MONITORING);
				// This call MUST be after SetState()
				ActivityMonitoring(FALSE);	// Reset Monitoring method
			END_IF
		END_IF

	E_RS_BASE_SUBSTATE.NOTOP_ERROR:			
		IF nEvent = E_SM_EVENT.HWOK THEN
			SetState(E_RS_BASE_STATE.NOTOP, E_RS_BASE_SUBSTATE.NOTOP_NOTREADY);
			RETURN;
		ELSIF nEvent = E_SM_EVENT.COMMOK THEN
			SetState(E_RS_BASE_STATE.NOTOP, nLastGoodSubstate);
			RETURN;			
		END_IF
		
	END_CASE

	(* Transitions from NOTOP state *)
	IF	nEvent = E_SM_EVENT.ERRHW OR
		nEvent = E_SM_EVENT.ERRCOMM	THEN
		ActionUnexpExecute();
		SetState(E_RS_BASE_STATE.NOTOP, E_RS_BASE_SUBSTATE.NOTOP_ERROR);
		RETURN;
	END_IF
	
//***********************************
// OPERATIONAL
//***********************************
E_RS_BASE_STATE.OP:

	(* Transitions from OP subastates *)
	CASE statRef.nSubstate OF
	E_RS_BASE_SUBSTATE.OP_ERROR:			
		IF nEvent = E_SM_EVENT.HWOK THEN
			SetStatus(E_SM_ERROR.OK, 'OK');
			SetState(E_RS_BASE_STATE.OP, E_RS_BASE_SUBSTATE.OP_IDLE);
			RETURN;			
		ELSIF nEvent = E_SM_EVENT.DISABLE THEN
			ActionDisableExecute();
			SetState(E_RS_BASE_STATE.NOTOP, E_RS_BASE_SUBSTATE.NOTOP_ERROR);
			RETURN;			
		ELSIF nEvent = E_SM_EVENT.COMMOK THEN
			SetState(E_RS_BASE_STATE.OP, nLastGoodSubstate);
			RETURN;			
		END_IF

	E_RS_BASE_SUBSTATE.OP_MONITORING:
		IF nEvent = E_SM_EVENT.DISABLE THEN
			ActionDisableExecute();
			RETURN;			
		ELSIF nEvent = E_SM_EVENT.STOPMON THEN
			ActionStopExecute();
			RETURN;			
		ELSIF nEvent = E_SM_EVENT.READDONE THEN
			SetState(E_RS_BASE_STATE.OP, E_RS_BASE_SUBSTATE.OP_IDLE);
			RETURN;			
		ELSIF nEvent = E_SM_EVENT.ERRCOMM THEN
			// Re-initialise on comm error.
			SetState(E_RS_BASE_STATE.NOTOP, E_RS_BASE_SUBSTATE.NOTOP_NOTREADY);
			RETURN;			
		END_IF
		
		
	E_RS_BASE_SUBSTATE.OP_IDLE:			
		IF nEvent = E_SM_EVENT.DISABLE THEN
			ActionDisableExecute();
			RETURN;			
		ELSIF nEvent = E_SM_EVENT.MONITOR OR nEvent = E_SM_EVENT.ENABLE THEN
			nReadType	:= E_RS_BASE_READ_TYPE.PERIODIC;
			ActivityMonitoring(FALSE);	// Reset Monitoring method
			SetState(E_RS_BASE_STATE.OP, E_RS_BASE_SUBSTATE.OP_MONITORING);
			RETURN;			
		END_IF
		
	END_CASE
	
	// Transitions from OP state.
	// Valid for any OP substate.
	IF nEvent = E_SM_EVENT.ERRHW THEN
		ActionUnexpExecute();
		SetState(E_RS_BASE_STATE.OP, E_RS_BASE_SUBSTATE.OP_ERROR);
		RETURN;
	ELSIF nEvent = E_SM_EVENT.ERRCOMM THEN
		SetState(E_RS_BASE_STATE.OP, E_RS_BASE_SUBSTATE.OP_ERROR);
		RETURN;
	END_IF
	
END_CASE

(* 
	"Global" internal transitions valid in any state should go here.
	They do not change the active state configuration. 
	They are evaluated after all the others transitions have been 
	considered.
*) 
IF nEvent = E_SM_EVENT.RESET THEN
	ActionResetExecute();
	SetState(E_RS_BASE_STATE.NOTOP, E_RS_BASE_SUBSTATE.NOTOP_NOTREADY);
	RETURN;
END_IF
END_METHOD

{attribute 'TcRpcEnable':='1'}
METHOD RPC_Disable : INT
VAR_INPUT
END_VAR
// RPC calls are not allowed in Local mode.
IF stat.bLocal THEN
	RPC_Disable	:= M_SetRpcStatus(E_SA_RPC_ERROR.LOCAL);
	RETURN;
END_IF

// Disable command is accepted only if device is in OP state.
IF stat.nState <> E_RS_BASE_STATE.OP THEN
	RPC_Disable	:= M_SetRpcStatus(E_SA_RPC_ERROR.NOT_OP);
	RETURN;
ELSE
	// Set disable command
	ctrl.nCommand := E_RS_COMMAND.DISABLE;
	ctrl.bExecute := TRUE;
	
	// Call was successful
	RPC_Disable	:= M_SetRpcStatus(E_SA_RPC_ERROR.OK);
END_IF
END_METHOD

{attribute 'TcRpcEnable':='1'}
METHOD RPC_Enable : INT
VAR_INPUT
END_VAR
// RPC calls are not allowed in Local mode.
IF stat.bLocal THEN
	RPC_Enable	:= M_SetRpcStatus(E_SA_RPC_ERROR.LOCAL);
	RETURN;
END_IF

// Enable command is accepted only if device is in NOTOP_READY.
IF	stat.nSubstate <> E_RS_BASE_SUBSTATE.NOTOP_READY		THEN
	RPC_Enable	:= M_SetRpcStatus(E_SA_RPC_ERROR.NOT_NOTOP_READY);
	RETURN;
ELSE
	// Set enable command
	ctrl.nCommand := E_RS_COMMAND.ENABLE;
	ctrl.bExecute := TRUE;
	
	// Call was successful
	RPC_Enable	:= M_SetRpcStatus(E_SA_RPC_ERROR.OK);
END_IF
END_METHOD

{attribute 'TcRpcEnable':='1'}
METHOD RPC_Init : INT
VAR_INPUT
END_VAR
// RPC calls are not allowed in Local mode.
IF stat.bLocal THEN
	RPC_Init	:= M_SetRpcStatus(E_SA_RPC_ERROR.LOCAL);
	RETURN;
END_IF


// Init command is accepted only if device is in NOTOP_NOTREADY or ERROR.
IF	stat.nSubstate <> E_RS_BASE_SUBSTATE.NOTOP_NOTREADY	AND  
	stat.nSubstate <> E_RS_BASE_SUBSTATE.NOTOP_ERROR		THEN
	RPC_Init	:= M_SetRpcStatus(E_SA_RPC_ERROR.NOT_NOTOP_NOTREADY);
	RETURN;
ELSE
	// Set INIT command
	ctrl.nCommand := E_RS_COMMAND.INIT;
	ctrl.bExecute := TRUE;
	
	// Call was successful
	RPC_Init	:= M_SetRpcStatus(E_SA_RPC_ERROR.OK);
END_IF
END_METHOD

{attribute 'TcRpcEnable':='1'}
METHOD RPC_Reset : INT
VAR_INPUT
END_VAR
// RPC calls are not allowed in Local mode.
IF stat.bLocal THEN
	RPC_Reset	:= M_SetRpcStatus(E_SA_RPC_ERROR.LOCAL);
	RETURN;
END_IF

ctrl.nCommand := E_RS_COMMAND.RESET;
ctrl.bExecute := TRUE;

// Call was successful
RPC_Reset	:= M_SetRpcStatus(E_SA_RPC_ERROR.OK);
END_METHOD

{attribute 'TcRpcEnable':='1'}
METHOD RPC_Stop : INT
VAR_INPUT
END_VAR
// RPC calls are not allowed in Local mode.
IF stat.bLocal THEN
	RPC_Stop	:= M_SetRpcStatus(E_SA_RPC_ERROR.LOCAL);
	RETURN;
END_IF

ctrl.nCommand := E_RS_COMMAND.STOP;
ctrl.bExecute := TRUE;

// Call was successful
RPC_Stop	:= M_SetRpcStatus(E_SA_RPC_ERROR.OK);
END_METHOD

END_FUNCTION_BLOCK

// ---- POUs/FB_SA_CHANNEL_BASE.TcPOU
FUNCTION_BLOCK FB_SA_CHANNEL_BASE
VAR_INPUT
END_VAR
VAR_OUTPUT
END_VAR
VAR
	{attribute 'OPC.UA.DA' := '1'}
	cfg:		T_SA_CH_CFG;	
	{attribute 'OPC.UA.DA' := '1'}
	ctrl:		T_SA_CH_CTRL;	

	{attribute 'OPC.UA.DA' := '1'}
	{attribute 'OPC.UA.DA.Access' := '1'}
	stat:		T_SA_CH_STATUS;	(* Common State Machine Status - ReadOnly *)

END_VAR

//
// The FB does not execute anything cyclically.
// It only executes method calls from instances of FB_SMAR_ACT_BASE.
//

METHOD M_Configure
VAR_INPUT
	in_sName:			STRING := 'Not Used'; 
	in_sUnits:			STRING := 'none';	// Positioner User Units
	// User scale. For example to use mm instead of m. m->mm (scale=0.001).
	// Pos [DevU] = lnScale * Pos [UU] / T_SA_CH_STATUS:nTUN_BASE_RES
	// Pos [UU]      = Pos [DevU] * T_SA_CH_STATUS:nTUN_BASE_RES / lnScale
	// [DevU] - Device units, i.e. pm or nd.
	// [UU] - User units, e.g. m, mm, deg, etc.
	in_lrScale:			LREAL := 1.0;			
	in_lrREF_POS:		LREAL := 0;			// Position of reference mark [UU]
	in_lrREF_VEL:		LREAL := 0.01;		// Velocity for referencing [UU/s]
	in_nHOLD:			DINT := -1;			// Hold time [ms]. -1 = infinite
	in_lrINP_THR:		LREAL := 0.01;		// In-position threshold [UU]	
	in_nINP_DEL:		UDINT := 1000;		// In-position delay [ms]
	in_lrMaxVelocity:	LREAL := 1.0;		// Maximum velocity	[UU]
	in_lrRangeLimitMin:	LREAL := 0.0;		// Lower SW Limit [UU}. Min=Max => no limit
	in_lrRangeLimitMax:	LREAL := 0.0;		// Upper SW Limit [UU]. Min=Max => no limit
	in_nREF_OPT:		UINT := 0;			// REFerencing in positive direction
	in_nCAL_OPT:		UINT := 0;			// CALibration in positive direction
	in_nPCON_OPT:		UINT := 256;		// Positioner control options. 256 - 'in-pos' flag set.
END_VAR
// Copy values to the config structure.
// This call sets initial config values but
// they can be overwritten from WS later on before
// sending the REF# command.
cfg.sName			:= in_sName;
cfg.sUnits			:= in_sUnits;
cfg.lrScale			:= in_lrScale;
cfg.lrREF_POS		:= in_lrREF_POS;
cfg.lrREF_VEL		:= in_lrREF_VEL;
cfg.nHOLD			:= in_nHOLD;
cfg.lrINP_THR		:= in_lrINP_THR;
cfg.nINP_DEL		:= in_nINP_DEL;
cfg.lrMaxVelocity	:= in_lrMaxVelocity;
cfg.lrRangeLimitMin	:= in_lrRangeLimitMin;
cfg.lrRangeLimitMax	:= in_lrRangeLimitMax;
cfg.nREF_OPT		:= in_nREF_OPT;
cfg.nCAL_OPT		:= in_nCAL_OPT;
cfg.nPCON_OPT		:= in_nPCON_OPT;

stat.bConfigured	:= TRUE;
END_METHOD

//
// Conversion from Device units [pm] or [nd] to user units, e.g. [mm] or [deg].
// This is a linear conversion.
// See also M_ConvertPosDev2User() for non-linear conversion of position.
//
METHOD M_ConvertDev2User : LREAL
VAR_INPUT
	lnDevValue:	LINT;
END_VAR
IF cfg.lrScale <> 0.0 THEN
	M_ConvertDev2User	:= LINT_TO_LREAL(lnDevValue) / cfg.lrScale * EXPT(10, stat.devStatus.nTUN_BASE_RES);
ELSE	
	M_ConvertDev2User	:= 0.0;
END_IF
END_METHOD

//
// Conversion position from Device units [pm] or [nd] to user units, e.g. mm or deg.
// By default, it is a linear conversion implemented in M_ConvertDev2User().
// However, the method can be overwritten to handle non-linear conversion.
//
METHOD M_ConvertPosDev2User : LREAL
VAR_INPUT
	lnDevValue:	LINT;
END_VAR
M_ConvertPosDev2User	:= M_ConvertDev2User(lnDevValue);
END_METHOD

//
// Conversion position from User Units, e.g. [mm] or [deg] to Device Units [pm] or [nd].
// By default, it is a linear conversion implemented in M_ConvertUser2Dev().
// However, the method can be overwritten to handle non-linear conversion.
//
METHOD M_ConvertPosUser2Dev : LINT
VAR_INPUT
	lrUserValue:	LREAL;
END_VAR
VAR
	lrVal:	LREAL;
END_VAR
M_ConvertPosUser2Dev	:= M_ConvertUser2Dev(lrUserValue);
END_METHOD

//
// Conversion from User Units, e.g. [mm] or [deg] to Device Units [pm] or [nd].
// This is a linear conversion.
// See also M_ConvertPosUser2Dev() for non-linear conversion of position.
//
METHOD M_ConvertUser2Dev : LINT
VAR_INPUT
	lrUserValue:	LREAL;
END_VAR
VAR
	lrVal:	LREAL;
END_VAR
// Convert UU to DevU as LREAL
lrVal	:= cfg.lrScale * lrUserValue / EXPT(10, stat.devStatus.nTUN_BASE_RES);
// Convert LREAL to LINT
M_ConvertUser2Dev	:= LREAL_TO_LINT(lrVal);
END_METHOD

// This is the only way for the positioner to know
// the status of the SmarAct MCS2 Controller that controls it.
METHOD M_GetCtrlState
VAR_INPUT
	bCtrlCommProblem:	BOOL;
	nCtrlErrorCode:		INT;
	nCtrlState:			INT;
END_VAR
stat.bCtrlCommProblem	:= bCtrlCommProblem;
stat.nCtrlErrorCode		:= nCtrlErrorCode;
stat.nCtrlState			:= nCtrlState;

//
// Set error if there is a problem with the MCS2 controller
// or the communication has been lost.
//
IF stat.bCtrlCommProblem	THEN
	stat.bError		:= TRUE;
	stat.nErrorCode	:= E_SA_CH_ERROR.COMM;
	stat.sErrorText	:= 'MCS2 Comm Problem';
	stat.sStatus	:= stat.sErrorText;
ELSIF stat.nCtrlErrorCode <> 0	THEN
	stat.bError		:= TRUE;
	stat.nErrorCode	:= E_SA_CH_ERROR.CTRL;
	stat.sErrorText	:= 'MCS2 Controller Problem';
	stat.sStatus	:= stat.sErrorText;
END_IF


//
// We cannot distinguish between unplugged cable and powered off MCS2 controller.
// If the communication is lost, go to NOTOP/NOT_READY.
//
IF stat.bCtrlCommProblem	THEN
	stat.bInitialised	:= FALSE;
	stat.nPosState		:= E_SA_POS_SM_STATE.NOT_READY;
	M_SetState(E_SA_POS_ELT_STATE.NOTOP);
	M_SetSubstate(E_SA_POS_ELT_SUBSTATE.NOTOP_ERROR);
END_IF
END_METHOD

METHOD M_GetErrorString : STRING
VAR_INPUT
END_VAR
IF	stat.stState.bRANGE_LIMIT_REACHED		THEN
	M_GetErrorString	:= 'ERROR: Range limit reached';
ELSIF	stat.stState.bEND_STOP_REACHED	THEN
	M_GetErrorString	:= 'ERROR: End Stop reached';
ELSIF	stat.stState.bFOLLOWING_LIMIT_REACHED	THEN
	M_GetErrorString	:= 'ERROR: Following error';
ELSIF	stat.stState.bPOSITIONER_OVERLOAD		THEN
	M_GetErrorString	:= 'ERROR: Positioner overload';
ELSIF	stat.stState.bOVER_TEMPERATURE			THEN
	M_GetErrorString	:= 'ERROR: Overtemperature';
ELSIF	stat.stState.bPOSITIONER_FAULT			THEN
	M_GetErrorString	:= 'ERROR: Positioner fault';
ELSIF	stat.stState.bMOVEMENT_FAILED			THEN
	M_GetErrorString	:= 'ERROR: Movement failed';
ELSE
	M_GetErrorString	:= 'Positioner Error';
END_IF
END_METHOD

METHOD M_GetModule : UINT
VAR_INPUT
END_VAR
M_GetModule	:= cfg.nMOD;
END_METHOD

METHOD M_SetChannel
VAR_INPUT
	index:	UINT;
END_VAR
// M_SetChannel() is called only for used channels

// Set the used flag
cfg.bUsed	:= TRUE;

// Set channel number, equal to the index.
cfg.nCHAN	:= index;

//
// MODule number that the channel belongs to [0..5].
// Calculated from the channel number. i.e. the index of this instance.
// channel = (Module x 3) + (CH-1)
// Module = index / 3
// index = 0, 1 or 2    => Module = 0
// index = 3, 4 or 5    => Module = 1
// ...
// index = 15, 16 or 17 => Module = 5
//
cfg.nMOD	:= index / 3;
END_METHOD

METHOD M_SetChanState
VAR_INPUT
	nStatus:	UDINT;	// Channel Status as UINT (WORD)
END_VAR
// Get Channel State as a number.
stat.nCH_STATE	:= nStatus;

//
// Extract Channel state from the status word.
//
stat.stState.bACTIVELY_MOVING			:= UDINT_TO_BOOL(nStatus AND E_SA_CH_STATE.BIT_ACTIVELY_MOVING);
stat.stState.bCLOSED_LOOP_ACTIVE		:= UDINT_TO_BOOL(nStatus AND E_SA_CH_STATE.BIT_CLOSED_LOOP_ACTIVE);
stat.stState.bCALIBRATING				:= UDINT_TO_BOOL(nStatus AND E_SA_CH_STATE.BIT_CALIBRATING);
stat.stState.bREFERENCING				:= UDINT_TO_BOOL(nStatus AND E_SA_CH_STATE.BIT_REFERENCING);
stat.stState.bMOVE_DELAYED				:= UDINT_TO_BOOL(nStatus AND E_SA_CH_STATE.BIT_MOVE_DELAYED);
stat.stState.bSENSOR_PRESENT			:= UDINT_TO_BOOL(nStatus AND E_SA_CH_STATE.BIT_SENSOR_PRESENT);
stat.stState.bIS_CALIBRATED				:= UDINT_TO_BOOL(nStatus AND E_SA_CH_STATE.BIT_IS_CALIBRATED);
stat.stState.bIS_REFERENCED				:= UDINT_TO_BOOL(nStatus AND E_SA_CH_STATE.BIT_IS_REFERENCED);
stat.stState.bEND_STOP_REACHED			:= UDINT_TO_BOOL(nStatus AND E_SA_CH_STATE.BIT_END_STOP_REACHED);
stat.stState.bRANGE_LIMIT_REACHED		:= UDINT_TO_BOOL(nStatus AND E_SA_CH_STATE.BIT_RANGE_LIMIT_REACHED);
stat.stState.bFOLLOWING_LIMIT_REACHED	:= UDINT_TO_BOOL(nStatus AND E_SA_CH_STATE.BIT_FOLLOWING_LIMIT_REACHED);
stat.stState.bMOVEMENT_FAILED			:= UDINT_TO_BOOL(nStatus AND E_SA_CH_STATE.BIT_MOVEMENT_FAILED);
stat.stState.bIS_STREAMING				:= UDINT_TO_BOOL(nStatus AND E_SA_CH_STATE.BIT_IS_STREAMING);
stat.stState.bPOSITIONER_OVERLOAD		:= UDINT_TO_BOOL(nStatus AND E_SA_CH_STATE.BIT_POSITIONER_OVERLOAD);
stat.stState.bOVER_TEMPERATURE			:= UDINT_TO_BOOL(nStatus AND E_SA_CH_STATE.BIT_OVER_TEMPERATURE);
stat.stState.bREFERENCE_MARK			:= UDINT_TO_BOOL(nStatus AND E_SA_CH_STATE.BIT_REFERENCE_MARK);
stat.stState.bIS_PHASED					:= UDINT_TO_BOOL(nStatus AND E_SA_CH_STATE.BIT_IS_PHASED);
stat.stState.bPOSITIONER_FAULT			:= UDINT_TO_BOOL(nStatus AND E_SA_CH_STATE.BIT_POSITIONER_FAULT);
stat.stState.bAMPLIFIER_ENABLED			:= UDINT_TO_BOOL(nStatus AND E_SA_CH_STATE.BIT_AMPLIFIER_ENABLED);
stat.stState.bIN_POSITION				:= UDINT_TO_BOOL(nStatus AND E_SA_CH_STATE.BIT_IN_POSITION);


IF	stat.stState.bRANGE_LIMIT_REACHED		OR
	stat.stState.bEND_STOP_REACHED			OR
	stat.stState.bFOLLOWING_LIMIT_REACHED	OR
	stat.stState.bMOVEMENT_FAILED			OR
	stat.stState.bPOSITIONER_OVERLOAD		OR
	stat.stState.bOVER_TEMPERATURE			OR
	stat.stState.bPOSITIONER_FAULT			THEN
		stat.stState.bERROR	:= TRUE;
		stat.bError			:= TRUE;
		stat.sErrorText		:= 'Positioner failure';
		stat.nPosState 		:= E_SA_POS_SM_STATE.ERROR;
ELSE
	// There is no positioner error but maybe the 
	// communication with the MCS2 controller is lost.
	stat.stState.bERROR	:= FALSE;
	
	// Check errors from the MCS2 controller.
	IF stat.bCtrlCommProblem  OR  stat.nCtrlErrorCode <> 0	THEN
		stat.bError	:= TRUE;
	ELSE
		stat.bError		:= FALSE;
		stat.nErrorCode	:= E_SA_CH_ERROR.OK;
		stat.sErrorText	:= 'OK';
	END_IF
END_IF
END_METHOD

METHOD M_SetCommandChannel : STRING
VAR_INPUT
	sCmd:	STRING;
END_VAR
VAR
	sCh:		STRING;
	sResult:	STRING;
	pos:		INT;
END_VAR
// Replace the hash (#) character in the command with a channel number.
// For example: Set Channel 3 in command ':CHAN#:TUN:BASE:UNIT?' 
//				Result = ':CHAN3:TUN:BASE:UNIT?'

// Find the position of the hash (#) character
pos	:= FIND(sCmd, '#');

IF pos > 0	THEN
	// Replace the hash (#) character with the channel number
	
	// Convert channel number into string.
	sCh	:= UINT_TO_STRING(cfg.nCHAN);
	
	// Create the resulting string that includes the channel number.
	sResult	:= REPLACE(sCmd, sCh, 1, pos);
ELSE
	// There was no hash (#) character in the command
	sResult	:= sCmd;
END_IF


M_SetCommandChannel	:= sResult;
END_METHOD

METHOD M_SetCommandModule : STRING
VAR_INPUT
	sCmd:	STRING;
END_VAR
VAR
	sMod:		STRING;
	sResult:	STRING;
	pos:		INT;
END_VAR
// Replace the hash (#) character in the command with a MODule number.
// For example: Set Module 3 in command ':MOD#:STAT?' 
//				Result = ':MOD3:STAT?'

// Find the position of the hash (#) character
pos	:= FIND(sCmd, '#');

IF pos > 0	THEN
	// Replace the hash (#) character with the module number
	
	// Convert module number into string.
	sMod	:= UINT_TO_STRING(cfg.nMOD);
	
	// Create the resulting string that includes the module number.
	sResult	:= REPLACE(sCmd, sMod, 1, pos);
ELSE
	// There was no hash (#) character in the command
	sResult	:= sCmd;
END_IF


M_SetCommandModule	:= sResult;
END_METHOD

METHOD M_SetCommandValue : STRING
VAR_INPUT
	sCmd:	STRING;
END_VAR
VAR
	sVal:		STRING;
	lrVal:		LREAL;
	lrVelo:		LREAL;
	lrPos:		LREAL;
	nVal:		DINT;
	lnVal:		LINT;
	sResult:	STRING;
	pos:		INT;
END_VAR
// Replace the '***' characters in the command with a value
// coming from the cfg structure.
// The value depends on the keyword.
// For example: Set value to 0 in command ':CHAN#:CAL:OPT ***' 
//				Result = ':CHAN#:CAL:OPT 0'

// Find the position of the '***' characters
pos	:= FIND(sCmd, '***');

IF pos > 0	THEN
	// Replace the hash *** characters with the corresponding value.
	// Check the command and take the value from the cfg.
	// Also, convert User Units [UU] to Device Units [DevU].
	IF FIND(sCmd, ':CAL:OPT') > 1	THEN
		sVal	:= UINT_TO_STRING(cfg.nCAL_OPT);
	ELSIF FIND(sCmd, ':REF:OPT') > 1	THEN
		sVal	:= UINT_TO_STRING(cfg.nREF_OPT);
	ELSIF FIND(sCmd, ':PCON:OPT') > 1	THEN
		sVal	:= UINT_TO_STRING(cfg.nPCON_OPT);
	ELSIF FIND(sCmd, ':HOLD') > 1	THEN
		sVal	:= DINT_TO_STRING(cfg.nHOLD);
	ELSIF FIND(sCmd, ':INP:THR') > 1	THEN
		// Convert LREAL to LINT to DINT.
		// Threshold must be positive.
		nVal	:= LINT_TO_DINT(ABS(M_ConvertUser2Dev(cfg.lrINP_THR)));
		// Convert DINT to STRING
		sVal	:= DINT_TO_STRING(nVal);
	ELSIF FIND(sCmd, ':INP:DEL') > 1	THEN
		sVal	:= UDINT_TO_STRING(cfg.nINP_DEL);
	ELSIF FIND(sCmd, ':RLIM:MIN') > 1	THEN
		// Convert LREAL to LINT
		lnVal	:= M_ConvertPosUser2Dev(cfg.lrRangeLimitMin);
		// Convert LINT to STRING
		sVal	:= LINT_TO_STRING(lnVal);
	ELSIF FIND(sCmd, ':RLIM:MAX') > 1	THEN
		// Convert LREAL to LINT
		lnVal	:= M_ConvertPosUser2Dev(cfg.lrRangeLimitMax);
		// Convert LINT to STRING
		sVal	:= LINT_TO_STRING(lnVal);
	ELSIF FIND(sCmd, ':POS ') > 1	THEN	// Note the space after POS !!!
		// Select correct position
		CASE stat.nPosState OF
			E_SA_POS_SM_STATE.CALIB_REF:
				lrPos	:= cfg.lrREF_POS;
			E_SA_POS_SM_STATE.MOVING:
				lrPos	:= ctrl.lrPos;
		END_CASE
		// Convert Pos in UU to DevU, i.e. LREAL to LINT
		lnVal	:= M_ConvertPosUser2Dev(lrPos);
		// In case we are calibrating the REFerence switch,
		// set/calibrate the actual position.
		IF stat.nPosState = E_SA_POS_SM_STATE.CALIB_REF	THEN
			stat.devStatus.lnPosActual	:= lnVal;
		END_IF
		// Convert LINT to STRING
		sVal	:= LINT_TO_STRING(lnVal);
	ELSIF FIND(sCmd, ':VEL ') > 1	THEN	// Note the space after POS !!!
		// Select correct velocity
		CASE stat.nPosState OF
			E_SA_POS_SM_STATE.INIT:
				lrVelo		:= cfg.lrREF_VEL;
				ctrl.lrVel	:= cfg.lrREF_VEL;
			E_SA_POS_SM_STATE.MOVING:
				lrVelo	:= ctrl.lrVel;
		END_CASE
		// Convert velocity in UU to DevU, i.e. LREAL to LINT.
		// Velocity must be positive.
		lnVal	:= ABS(M_ConvertUser2Dev(lrVelo));
		// Convert LINT to STRING
		sVal	:= LINT_TO_STRING(lnVal);
	ELSIF FIND(sCmd, ':MOVE') = 1	THEN	// Note =1 !!!, cmd starts with ':MOVE'
		// Convert target position from UU to DevU, i.e. LREAL to LINT
		lnVal	:= M_ConvertPosUser2Dev(ctrl.lrPos);
		// Convert LINT to STRING
		sVal	:= LINT_TO_STRING(lnVal);
	ELSE
		M_SetCommandValue	:= sCmd;
		RETURN;
	END_IF
	
	// Create the resulting string that includes the value.
	// Replace 3 characters '***' starting from pos with the value.
	sResult	:= REPLACE(sCmd, sVal, 3, pos);
ELSE
	// There was no hash (#) character in the command
	sResult	:= sCmd;
END_IF


M_SetCommandValue	:= sResult;
END_METHOD

//
// Set next positioner State Machine State.
// This is done at the end of command list execution.
// It Returns TRUE if the state has changed.
//
METHOD M_SetNextPosState : BOOL
VAR_INPUT
END_VAR
CASE stat.nPosState OF
	E_SA_POS_SM_STATE.NOT_READY:
		IF ctrl.nCmd = E_SA_CH_CMD.CALIB	THEN
			ctrl.nCmd 			:= E_SA_CH_CMD.NONE;	// Reset command
			stat.nPosState 		:= E_SA_POS_SM_STATE.CALIB;
			stat.bInitialised	:= FALSE;
			stat.sStatus		:= 'Calibrating...';
			M_SetState(E_SA_POS_ELT_STATE.NOTOP);
			M_SetSubstate(E_SA_POS_ELT_SUBSTATE.NOTOP_INITIALIZING);
			M_SetNextPosState	:= TRUE;	// State HAS changed
		ELSIF ctrl.nCmd = E_SA_CH_CMD.REF	THEN
			ctrl.nCmd 			:= E_SA_CH_CMD.NONE;	// Reset command
			stat.nPosState 		:= E_SA_POS_SM_STATE.INIT;
			stat.sStatus		:= 'Referencing/INIT Started';
			M_SetState(E_SA_POS_ELT_STATE.NOTOP);
			M_SetSubstate(E_SA_POS_ELT_SUBSTATE.NOTOP_INITIALIZING);
			M_SetNextPosState	:= TRUE;	// State HAS changed
		ELSE
			M_SetNextPosState	:= FALSE;	// State has NOT changed
		END_IF
	E_SA_POS_SM_STATE.CALIB:
		stat.nPosState := E_SA_POS_SM_STATE.NOT_READY;
		stat.bInitialised	:= FALSE;
		stat.sStatus		:= 'Calibration completed';
		M_SetNextPosState	:= TRUE;	// State HAS changed
	E_SA_POS_SM_STATE.INIT:
		stat.nPosState := E_SA_POS_SM_STATE.POST_INIT;
		stat.sStatus		:= 'Updating configuration...';
		M_SetNextPosState	:= TRUE;	// State HAS changed
	E_SA_POS_SM_STATE.POST_INIT:
		IF ctrl.nCmd = E_SA_CH_CMD.STOP	THEN
			ctrl.nCmd 			:= E_SA_CH_CMD.NONE;	// Reset command
			stat.nPosState 		:= E_SA_POS_SM_STATE.STOP;
			stat.sStatus		:= 'Stopping...';
			M_SetNextPosState	:= TRUE;	// State HAS changed
		ELSIF	NOT stat.stState.bACTIVELY_MOVING	AND
				stat.stState.bIS_REFERENCED			AND
				stat.stState.bIN_POSITION			AND
				stat.stState.bREFERENCE_MARK			THEN
			stat.nPosState := E_SA_POS_SM_STATE.CALIB_REF;
			stat.sStatus		:= 'Referencing completed';
			M_SetNextPosState	:= TRUE;	// State HAS changed
		ELSE
			stat.sStatus		:= 'Referencing/Initialising...';
			M_SetNextPosState	:= FALSE;	// State has NOT changed
		END_IF
	E_SA_POS_SM_STATE.CALIB_REF:
		stat.nPosState 	:= E_SA_POS_SM_STATE.READY;	// was OP
		stat.nLastPosState := E_SA_POS_SM_STATE.CALIB_REF;
		stat.bInitialised	:= TRUE;
		stat.sStatus		:= 'Reference mark calibrated - initialised';
		M_SetNextPosState	:= TRUE;	// State HAS changed
	E_SA_POS_SM_STATE.READY:
		IF ctrl.nCmd = E_SA_CH_CMD.ENABLE	THEN
			ctrl.nCmd 			:= E_SA_CH_CMD.NONE;	// Reset command
			stat.nPosState 		:= E_SA_POS_SM_STATE.OP;
			stat.sStatus		:= 'Operational';
			M_SetState(E_SA_POS_ELT_STATE.OP);
			M_SetSubstate(E_SA_POS_ELT_SUBSTATE.OP_STANDSTILL);
			M_SetNextPosState	:= TRUE;	// State HAS changed
		ELSIF ctrl.nCmd = E_SA_CH_CMD.RESET	THEN
			ctrl.nCmd 			:= E_SA_CH_CMD.NONE;	// Reset command
			stat.nPosState 		:= E_SA_POS_SM_STATE.NOT_READY;
			stat.bInitialised	:= FALSE;
			stat.nErrorCode		:= E_SA_CH_ERROR.OK; 
			stat.sErrorText		:= 'OK';
			stat.sStatus		:= 'Positioner Reset';
			M_SetState(E_SA_POS_ELT_STATE.NOTOP);
			M_SetSubstate(E_SA_POS_ELT_SUBSTATE.NOTOP_NOTREADY);
			M_SetNextPosState	:= TRUE;	// State HAS changed
		ELSE
			M_SetNextPosState	:= FALSE;	// State has NOT changed
		END_IF
	E_SA_POS_SM_STATE.OP:
		IF ctrl.nCmd = E_SA_CH_CMD.RESET	THEN
			ctrl.nCmd 			:= E_SA_CH_CMD.NONE;	// Reset command
			stat.nPosState 		:= E_SA_POS_SM_STATE.NOT_READY;
			stat.bInitialised	:= FALSE;
			stat.nErrorCode		:= E_SA_CH_ERROR.OK; 
			stat.sErrorText		:= 'OK';
			stat.sStatus		:= 'Positioner Reset';
			M_SetState(E_SA_POS_ELT_STATE.NOTOP);
			M_SetSubstate(E_SA_POS_ELT_SUBSTATE.NOTOP_NOTREADY);
			M_SetNextPosState	:= TRUE;	// State HAS changed
		ELSIF ctrl.nCmd = E_SA_CH_CMD.DISABLE	THEN
			ctrl.nCmd 			:= E_SA_CH_CMD.NONE;	// Reset command
			stat.nPosState 		:= E_SA_POS_SM_STATE.READY;
			stat.sStatus		:= 'Ready';
			M_SetState(E_SA_POS_ELT_STATE.NOTOP);
			M_SetSubstate(E_SA_POS_ELT_SUBSTATE.NOTOP_READY);
			M_SetNextPosState	:= TRUE;	// State HAS changed
		ELSIF ctrl.nCmd = E_SA_CH_CMD.MOV	THEN
			ctrl.nCmd 			:= E_SA_CH_CMD.NONE;	// Reset command
			stat.stState.bACTIVELY_MOVING	:= TRUE;
			stat.stState.bIN_POSITION		:= FALSE;
			stat.nPosState 		:= E_SA_POS_SM_STATE.MOVING;
			stat.nLastPosState 	:= E_SA_POS_SM_STATE.OP;
			stat.sStatus		:= 'Moving...';
			M_SetSubstate(E_SA_POS_ELT_SUBSTATE.OP_MOVING);
			M_SetNextPosState	:= TRUE;	// State HAS changed
		ELSIF ctrl.nCmd = E_SA_CH_CMD.STOP	THEN
			ctrl.nCmd 			:= E_SA_CH_CMD.NONE;	// Reset command
			stat.nPosState 		:= E_SA_POS_SM_STATE.STOP;
			stat.sStatus		:= 'Stopping...';
			M_SetSubstate(E_SA_POS_ELT_SUBSTATE.OP_STOPPING);
			M_SetNextPosState	:= TRUE;	// State HAS changed
		ELSIF	NOT stat.stState.bACTIVELY_MOVING	AND
				stat.stState.bIN_POSITION			AND
				stat.nLastPosState <> E_SA_POS_SM_STATE.CALIB_REF	THEN
					stat.sStatus		:= 'Move completed';
					M_SetNextPosState	:= FALSE;	// State has NOT changed
		ELSE
			M_SetNextPosState	:= FALSE;	// State has NOT changed
		END_IF
	E_SA_POS_SM_STATE.MOVING:
		IF ctrl.nCmd = E_SA_CH_CMD.STOP	THEN
			ctrl.nCmd 			:= E_SA_CH_CMD.NONE;	// Reset command
			stat.nPosState 		:= E_SA_POS_SM_STATE.STOP;
			stat.sStatus		:= 'Stopping...';
			M_SetSubstate(E_SA_POS_ELT_SUBSTATE.OP_STOPPING);
			M_SetNextPosState	:= TRUE;	// State HAS changed
		ELSE
			stat.nPosState := E_SA_POS_SM_STATE.OP;
			M_SetNextPosState	:= TRUE;	// State HAS changed
		END_IF
	E_SA_POS_SM_STATE.STOP:
		stat.nPosState := E_SA_POS_SM_STATE.OP;
		stat.sStatus		:= 'Positioner Stopped';
		M_SetNextPosState	:= TRUE;	// State HAS changed
	E_SA_POS_SM_STATE.ERROR:
		IF ctrl.nCmd = E_SA_CH_CMD.CALIB	THEN
			ctrl.nCmd 			:= E_SA_CH_CMD.NONE;	// Reset command
			stat.nPosState 		:= E_SA_POS_SM_STATE.CALIB;
			stat.bInitialised	:= FALSE;
			stat.sStatus		:= 'Calibrating...';
			M_SetState(E_SA_POS_ELT_STATE.NOTOP);
			M_SetSubstate(E_SA_POS_ELT_SUBSTATE.NOTOP_NOTREADY);
			M_SetNextPosState	:= TRUE;	// State HAS changed
		ELSIF ctrl.nCmd = E_SA_CH_CMD.REF	THEN
			ctrl.nCmd 			:= E_SA_CH_CMD.NONE;	// Reset command
			stat.nPosState 		:= E_SA_POS_SM_STATE.INIT;
			stat.bInitialised	:= FALSE;
			stat.sStatus		:= 'Referencing/INIT Started';
			M_SetState(E_SA_POS_ELT_STATE.NOTOP);
			M_SetSubstate(E_SA_POS_ELT_SUBSTATE.NOTOP_NOTREADY);
			M_SetNextPosState	:= TRUE;	// State HAS changed
		ELSIF ctrl.nCmd = E_SA_CH_CMD.MOV	THEN
			ctrl.nCmd 			:= E_SA_CH_CMD.NONE;	// Reset command
			stat.stState.bACTIVELY_MOVING	:= TRUE;
			stat.stState.bIN_POSITION		:= FALSE;
			stat.nPosState 		:= E_SA_POS_SM_STATE.MOVING;
			stat.nLastPosState 	:= E_SA_POS_SM_STATE.OP;
			stat.sStatus		:= 'Moving...';
			M_SetSubstate(E_SA_POS_ELT_SUBSTATE.OP_MOVING);
			M_SetNextPosState	:= TRUE;	// State HAS changed
		ELSIF ctrl.nCmd = E_SA_CH_CMD.RESET	THEN
			ctrl.nCmd 			:= E_SA_CH_CMD.NONE;	// Reset command
			stat.nPosState 		:= E_SA_POS_SM_STATE.NOT_READY;
			stat.bInitialised	:= FALSE;
			stat.nErrorCode		:= E_SA_CH_ERROR.OK; 
			stat.sErrorText		:= 'OK';
			stat.sStatus		:= 'Positioner Reset';
			M_SetState(E_SA_POS_ELT_STATE.NOTOP);
			M_SetSubstate(E_SA_POS_ELT_SUBSTATE.NOTOP_NOTREADY);
			M_SetNextPosState	:= TRUE;	// State HAS changed
		ELSE
			stat.sStatus		:= M_GetErrorString();
			M_SetNextPosState	:= FALSE;	// State has NOT changed
		END_IF
END_CASE
END_METHOD

METHOD M_SetRpcStatus : INT
VAR_INPUT
	nErrorCode:	INT;
END_VAR
stat.nRpcErrorCode	:= nErrorCode;
stat.sRpcErrorText	:= F_GetRpcErrorText(nErrorCode);

M_SetRpcStatus	:= nErrorCode;
END_METHOD

METHOD M_SetState
VAR_INPUT
	nState: E_SA_POS_ELT_STATE;
END_VAR
stat.nState	:= nState;

// Set substate string
CASE nState	OF
	E_SA_POS_ELT_STATE.NOTOP: 	stat.sState	:= 'NOT OP';
	E_SA_POS_ELT_STATE.OP: 		stat.sState	:= 'OPERATIONAL';
END_CASE
END_METHOD

METHOD M_SetSubstate
VAR_INPUT
	nSubstate: E_SA_POS_ELT_SUBSTATE;
END_VAR
stat.nSubstate	:= nSubstate;

// Set substate string
CASE nSubstate	OF
	E_SA_POS_ELT_SUBSTATE.NOTOP_NOTREADY: 		
		stat.sSubstate	:= 'NOT READY';
		stat.sStatus	:= '';
	E_SA_POS_ELT_SUBSTATE.NOTOP_READY: 			stat.sSubstate	:= 'READY';
	E_SA_POS_ELT_SUBSTATE.NOTOP_INITIALIZING:	stat.sSubstate	:= 'INITIALIZING';
	E_SA_POS_ELT_SUBSTATE.NOTOP_ABORTING:		stat.sSubstate	:= 'ABORTING';
	E_SA_POS_ELT_SUBSTATE.NOTOP_ERROR:			stat.sSubstate	:= 'ERROR';
	
	E_SA_POS_ELT_SUBSTATE.OP_STANDSTILL:		stat.sSubstate	:= 'STANDSTILL';            
	E_SA_POS_ELT_SUBSTATE.OP_MOVING:			stat.sSubstate	:= 'MOVING';
	E_SA_POS_ELT_SUBSTATE.OP_SETTING_POS:		stat.sSubstate	:= 'SETTING POS';
	E_SA_POS_ELT_SUBSTATE.OP_STOPPING:			stat.sSubstate	:= 'STOPPING';
	E_SA_POS_ELT_SUBSTATE.OP_ERROR:				stat.sSubstate	:= 'ERROR';
	
END_CASE
END_METHOD

//
// Convert Positioner status from Device to User mode.
//
METHOD M_UpdateStatus
VAR_INPUT
END_VAR
//
// Update bEnabled flag.
// If TRUE, it means that the amplifier is enabled and the sensor is present.
//
stat.bEnabled	:= stat.stState.bAMPLIFIER_ENABLED AND  stat.stState.bSENSOR_PRESENT;


//
// Set the in-position flag
//
stat.bInPosition	:= stat.stState.bIN_POSITION;


//
// Set target and actual positions in [UU]
//
stat.lrPosTarget	:= M_ConvertPosDev2User(stat.devStatus.lnPosTarget);
stat.lrPosActual	:= M_ConvertPosDev2User(stat.devStatus.lnPosActual);


//
// Set Standard ELT States and Substates
//


//
// Substate
//
CASE stat.nState OF
	E_SA_POS_ELT_STATE.NOTOP:
	/////////////////////////
	IF stat.bError	THEN
		M_SetSubstate(E_SA_POS_ELT_SUBSTATE.NOTOP_ERROR);
	ELSIF	stat.nPosState = E_SA_POS_SM_STATE.NOT_READY	THEN
		M_SetSubstate(E_SA_POS_ELT_SUBSTATE.NOTOP_NOTREADY);
	ELSIF 	stat.nPosState = E_SA_POS_SM_STATE.CALIB  		OR
			stat.nPosState = E_SA_POS_SM_STATE.INIT  		OR
			stat.nPosState = E_SA_POS_SM_STATE.POST_INIT	OR	
			stat.nPosState = E_SA_POS_SM_STATE.CALIB_REF  		THEN
		M_SetSubstate(E_SA_POS_ELT_SUBSTATE.NOTOP_INITIALIZING);
	ELSIF 	stat.nPosState = E_SA_POS_SM_STATE.READY  	THEN
		M_SetSubstate(E_SA_POS_ELT_SUBSTATE.NOTOP_READY);
	ELSE
		M_SetSubstate(E_SA_POS_ELT_SUBSTATE.NOTOP_NOTREADY);
	END_IF
	
	E_SA_POS_ELT_STATE.OP:
	//////////////////////
	IF stat.stState.bACTIVELY_MOVING	THEN
		IF stat.nPosState = E_SA_POS_SM_STATE.STOP	THEN
			M_SetSubstate(E_SA_POS_ELT_SUBSTATE.OP_STOPPING);
		ELSE
			M_SetSubstate(E_SA_POS_ELT_SUBSTATE.OP_MOVING);
		END_IF
	ELSIF stat.stState.bERROR	THEN
		M_SetSubstate(E_SA_POS_ELT_SUBSTATE.OP_ERROR);
	ELSE
		M_SetSubstate(E_SA_POS_ELT_SUBSTATE.OP_STANDSTILL);
	END_IF
END_CASE
END_METHOD

{attribute 'TcRpcEnable':='1'}
METHOD RPC_Disable : INT
VAR_INPUT
END_VAR
// If the SmarAct MCS2 Controller is in error,
// the positioner cannot be controlled.
IF stat.nCtrlErrorCode <> 0  OR  stat.nCtrlState <> E_RS_BASE_STATE.OP THEN
	RPC_Disable	:= M_SetRpcStatus(E_SA_RPC_ERROR.CTRL_ERROR);
	RETURN;
END_IF


// RPC calls are not allowed in Local mode.
IF stat.bLocal THEN
	RPC_Disable	:= M_SetRpcStatus(E_SA_RPC_ERROR.LOCAL);
	RETURN;
END_IF

// Disable command is accepted only if device is in OP state.
IF stat.nState <> E_SA_POS_ELT_STATE.OP THEN
	RPC_Disable	:= M_SetRpcStatus(E_SA_RPC_ERROR.NOT_OP);
	RETURN;
END_IF

// Set DISABLE command
ctrl.nCmd	:= E_SA_CH_CMD.DISABLE;

// Call was successful
RPC_Disable	:= M_SetRpcStatus(E_SA_RPC_ERROR.OK);
END_METHOD

{attribute 'TcRpcEnable':='1'}
METHOD RPC_Enable : INT
VAR_INPUT
END_VAR
// If the SmarAct MCS2 Controller is in error,
// the positioner cannot be controlled.
IF stat.nCtrlErrorCode <> 0  OR  stat.nCtrlState <> E_RS_BASE_STATE.OP THEN
	RPC_Enable	:= M_SetRpcStatus(E_SA_RPC_ERROR.CTRL_ERROR);
	RETURN;
END_IF


// RPC calls are not allowed in Local mode.
IF stat.bLocal THEN
	RPC_Enable	:= M_SetRpcStatus(E_SA_RPC_ERROR.LOCAL);
	RETURN;
END_IF

// Enable command is accepted only if device is NOT OPERATIONAL.
IF	stat.nState <> E_SA_POS_ELT_STATE.NOTOP		THEN
	RPC_Enable	:= M_SetRpcStatus(E_SA_RPC_ERROR.NOT_NOTOP_READY);
	RETURN;
END_IF


// Set ENABLE command
ctrl.nCmd	:= E_SA_CH_CMD.ENABLE;

// Call was successful
RPC_Enable	:= M_SetRpcStatus(E_SA_RPC_ERROR.OK);
END_METHOD

{attribute 'TcRpcEnable':='1'}
METHOD RPC_Init : INT
VAR_INPUT
END_VAR
//
// REFerencing of SmarAct Positioner is equivalent to Motor INIT.
//

// If the SmarAct MCS2 Controller is in error,
// the positioner cannot be controlled.
IF stat.nCtrlErrorCode <> 0  OR  stat.nCtrlState <> E_RS_BASE_STATE.OP THEN
	RPC_Init	:= M_SetRpcStatus(E_SA_RPC_ERROR.CTRL_ERROR);
	RETURN;
END_IF


// RPC calls are not allowed in Local mode.
IF stat.bLocal THEN
	RPC_Init	:= M_SetRpcStatus(E_SA_RPC_ERROR.LOCAL);
	RETURN;
END_IF


// Set INIT (REF#) command
ctrl.nCmd	:= E_SA_CH_CMD.REF;

// Call was successful
RPC_Init	:= M_SetRpcStatus(E_SA_RPC_ERROR.OK);
END_METHOD

{attribute 'TcRpcEnable':='1'}
METHOD RPC_MoveAbs : INT
VAR_INPUT
	in_lrPos:		LREAL;	// Target position [UU]
	in_lrVel:		LREAL;	// Target velocity [UU/s]
END_VAR
// If the SmarAct MCS2 Controller is in error,
// the positioner cannot be controlled.
IF stat.nCtrlErrorCode <> 0  OR  stat.nCtrlState <> E_RS_BASE_STATE.OP THEN
	RPC_MoveAbs	:= M_SetRpcStatus(E_SA_RPC_ERROR.CTRL_ERROR);
	RETURN;
END_IF


// RPC calls are not allowed in Local mode.
IF stat.bLocal THEN
	RPC_MoveAbs	:= M_SetRpcStatus(E_SA_RPC_ERROR.LOCAL);
	RETURN;
// Move Absolute command is accepted only in OP state.
ELSIF	stat.nState <> E_SA_POS_ELT_STATE.OP	THEN
	RPC_MoveAbs	:= M_SetRpcStatus(E_SA_RPC_ERROR.NOT_OP);
	RETURN;
// The positioner has to be initialised / OP (operational), i.e. already REFerenced.
ELSIF	NOT stat.bInitialised	THEN
	RPC_MoveAbs	:= M_SetRpcStatus(E_SA_RPC_ERROR.CH_NOT_OP);
	RETURN;
// Set velocity cannot be 0.0.
ELSIF	in_lrVel = 0.0	THEN
	RPC_MoveAbs	:= M_SetRpcStatus(E_SA_RPC_ERROR.VEL_ZERO);
	RETURN;
// Set velocity cannot be < 0.0.
ELSIF	in_lrVel <= 0.0	THEN
	RPC_MoveAbs	:= M_SetRpcStatus(E_SA_RPC_ERROR.VEL_NEG);
	RETURN;
// Set velocity cannot be greater than MAX Velocity.
ELSIF	in_lrVel > cfg.lrMaxVelocity	THEN
	RPC_MoveAbs	:= M_SetRpcStatus(E_SA_RPC_ERROR.VEL_MAX);
	RETURN;
// If SW limits are active, check the limits
ELSIF cfg.lrRangeLimitMax > cfg.lrRangeLimitMin THEN
	IF in_lrPos < cfg.lrRangeLimitMin THEN
		RPC_MoveAbs	:= M_SetRpcStatus(E_SA_RPC_ERROR.SW_LIMIT_LOWER);
		RETURN;
	ELSIF in_lrPos > cfg.lrRangeLimitMax THEN
		RPC_MoveAbs	:= M_SetRpcStatus(E_SA_RPC_ERROR.SW_LIMIT_UPPER);
		RETURN;
	END_IF
END_IF

// Set command
ctrl.nCmd	:= E_SA_CH_CMD.MOV;
ctrl.lrPos	:= in_lrPos;
ctrl.lrVel	:= in_lrVel;


// Call was successful
RPC_MoveAbs	:= M_SetRpcStatus(E_SA_RPC_ERROR.OK);
END_METHOD

{attribute 'TcRpcEnable':='1'}
METHOD RPC_MoveRel : INT
VAR_INPUT
	in_lrPos:		LREAL;	// Target relative position [UU]
	in_lrVel:		LREAL;	// Target velocity [UU/s]
END_VAR
VAR
	lrPos:			LREAL;	// New absolute position [UU]
END_VAR
// If the SmarAct MCS2 Controller is in error,
// the positioner cannot be controlled.
IF stat.nCtrlErrorCode <> 0  OR  stat.nCtrlState <> E_RS_BASE_STATE.OP THEN
	RPC_MoveRel	:= M_SetRpcStatus(E_SA_RPC_ERROR.CTRL_ERROR);
	RETURN;
END_IF


// Get new absolute position
lrPos	:= stat.lrPosActual + in_lrPos;

